SPLINE
SPL {X  -150.342, Y  +330.952, Z    +0.000, E1   +71.154, E3 +35565.120}
SPL {X  -141.358, Y  +310.748, Z    +0.000, E1   +71.233, E3 +35577.826}
SPL {X  -134.330, Y  +298.778, Z    +0.000, E1   +70.323, E3 +35591.673}
SPL {X  -128.957, Y  +290.989, Z    +0.000, E1   +69.528, E3 +35601.038}
SPL {X  -124.846, Y  +285.632, Z    +0.000, E1   +68.906, E3 +35607.502}
SPL {X  -121.783, Y  +281.927, Z    +0.000, E1   +68.403, E3 +35611.934}
SPL {X   -79.219, Y  +246.688, Z    +0.000, E1   +55.887, E3 +35733.440}
ENDSPLINE

SPLINE
SPL {X  -125.038, Y  +285.873, Z    +0.000, E1   +53.023, E3 +35910.481}
SPL {X  -149.949, Y  +329.886, Z    +0.000, E1   +41.515, E3 +35932.046}
SPL {X  -157.246, Y  +356.141, Z    +0.000, E1   +27.282, E3 +35937.103}
SPL {X  -159.525, Y  +373.376, Z    +0.000, E1   +13.812, E3 +35938.760}
SPL {X  -160.000, Y  +387.264, Z    +0.000, E1    +0.544, E3 +35939.218}
SPL {X  -160.000, Y  +390.384, Z    +0.000, E1    -6.008, E3 +35939.255}
SPL {X  -160.000, Y  +395.752, Z    +0.000, E1   -19.038, E3 +35939.449}
SPL {X  -160.000, Y  +404.289, Z    +0.000, E1   -38.292, E3 +35940.117}
SPL {X  -160.000, Y  +418.681, Z    +0.000, E1   -56.949, E3 +35942.307}
SPL {X  -160.000, Y  +471.977, Z    +0.000, E1   -70.792, E3 +35958.826}
SPL {X  -159.977, Y  +677.138, Z    +0.000, E1   -73.665, E3 +36055.317}
SPL {X  -157.805, Y  +700.810, Z    +0.000, E1   -73.511, E3 +36072.147}
SPL {X  -152.242, Y  +723.618, Z    +0.000, E1   -72.940, E3 +36092.060}
SPL {X  -145.929, Y  +740.010, Z    +0.000, E1   -72.229, E3 +36108.532}
SPL {X  -139.114, Y  +753.439, Z    +0.000, E1   -71.436, E3 +36123.170}
SPL {X  -132.333, Y  +764.333, Z    +0.000, E1   -70.535, E3 +36135.794}
SPL {X  -125.486, Y  +773.664, Z    +0.000, E1   -69.598, E3 +36146.768}
SPL {X  -121.321, Y  +778.713, Z    +0.000, E1   -68.872, E3 +36152.778}
SPL {X   -77.337, Y  +814.468, Z    +0.000, E1   -56.377, E3 +36271.410}
ENDSPLINE

SPLINE
SPL {X  -134.727, Y  +760.706, Z    +0.000, E1   -50.460, E3 +36459.641}
SPL {X  -155.580, Y  +711.748, Z    +0.000, E1   -32.084, E3 +36476.556}
SPL {X  -159.445, Y  +687.715, Z    +0.000, E1   -14.660, E3 +36479.403}
SPL {X  -159.995, Y  +675.725, Z    +0.000, E1    -3.424, E3 +36479.914}
SPL {X  -160.000, Y  +671.714, Z    +0.000, E1    +0.835, E3 +36479.954}
SPL {X  -160.000, Y  +663.084, Z    +0.000, E1   +21.134, E3 +36480.278}
SPL {X  -160.000, Y  +650.910, Z    +0.000, E1   +46.005, E3 +36481.432}
SPL {X  -160.000, Y  +634.843, Z    +0.000, E1   +61.273, E3 +36484.109}
SPL {X  -160.000, Y  +578.679, Z    +0.000, E1   +71.665, E3 +36501.943}
SPL {X  -160.000, Y  +387.528, Z    +0.000, E1   +73.487, E3 +36594.755}
SPL {X  -159.218, Y  +369.903, Z    +0.000, E1   +73.425, E3 +36606.622}
SPL {X  -156.808, Y  +353.900, Z    +0.000, E1   +73.180, E3 +36619.226}
SPL {X  -154.539, Y  +344.254, Z    +0.000, E1   +72.827, E3 +36628.763}
ENDSPLINE

SPLINE
SPL {X  -157.258, Y  +356.206, Z    +0.000, E1   +70.434, E3 +36643.336}
ENDSPLINE

SPLINE
SPL {X  -150.342, Y  +330.952, Z    +0.000, E1   +71.154, E3 +36655.008}
SPL {X  -141.358, Y  +310.748, Z    +0.000, E1   +71.233, E3 +36667.714}
SPL {X  -134.330, Y  +298.778, Z    +0.000, E1   +70.323, E3 +36681.561}
SPL {X  -128.957, Y  +290.989, Z    +0.000, E1   +69.528, E3 +36690.926}
SPL {X  -124.846, Y  +285.632, Z    +0.000, E1   +68.906, E3 +36697.390}
SPL {X  -121.783, Y  +281.927, Z    +0.000, E1   +68.403, E3 +36701.822}
SPL {X   -79.219, Y  +246.688, Z    +0.000, E1   +55.887, E3 +36823.328}
ENDSPLINE

SPLINE
SPL {X  -125.038, Y  +285.873, Z    +0.000, E1   +53.023, E3 +37000.369}
SPL {X  -149.949, Y  +329.886, Z    +0.000, E1   +41.515, E3 +37021.934}
SPL {X  -157.246, Y  +356.141, Z    +0.000, E1   +27.282, E3 +37026.991}
SPL {X  -159.525, Y  +373.376, Z    +0.000, E1   +13.812, E3 +37028.648}
SPL {X  -160.000, Y  +387.264, Z    +0.000, E1    +0.544, E3 +37029.106}
SPL {X  -160.000, Y  +390.384, Z    +0.000, E1    -6.008, E3 +37029.143}
SPL {X  -160.000, Y  +395.752, Z    +0.000, E1   -19.038, E3 +37029.337}
SPL {X  -160.000, Y  +404.289, Z    +0.000, E1   -38.292, E3 +37030.005}
SPL {X  -160.000, Y  +418.681, Z    +0.000, E1   -56.949, E3 +37032.195}
SPL {X  -160.000, Y  +471.977, Z    +0.000, E1   -70.792, E3 +37048.714}
SPL {X  -159.977, Y  +677.138, Z    +0.000, E1   -73.665, E3 +37145.205}
SPL {X  -157.805, Y  +700.810, Z    +0.000, E1   -73.511, E3 +37162.035}
SPL {X  -152.242, Y  +723.618, Z    +0.000, E1   -72.940, E3 +37181.948}
SPL {X  -145.929, Y  +740.010, Z    +0.000, E1   -72.229, E3 +37198.420}
SPL {X  -139.114, Y  +753.439, Z    +0.000, E1   -71.436, E3 +37213.058}
SPL {X  -132.333, Y  +764.333, Z    +0.000, E1   -70.535, E3 +37225.682}
SPL {X  -125.486, Y  +773.664, Z    +0.000, E1   -69.598, E3 +37236.656}
SPL {X  -121.321, Y  +778.713, Z    +0.000, E1   -68.872, E3 +37242.666}
SPL {X   -77.337, Y  +814.468, Z    +0.000, E1   -56.377, E3 +37361.298}
ENDSPLINE

SPLINE
SPL {X  -134.727, Y  +760.706, Z    +0.000, E1   -50.460, E3 +37549.529}
SPL {X  -155.580, Y  +711.748, Z    +0.000, E1   -32.084, E3 +37566.444}
SPL {X  -159.445, Y  +687.715, Z    +0.000, E1   -14.660, E3 +37569.291}
SPL {X  -159.995, Y  +675.725, Z    +0.000, E1    -3.424, E3 +37569.802}
SPL {X  -160.000, Y  +671.714, Z    +0.000, E1    +0.835, E3 +37569.842}
SPL {X  -160.000, Y  +663.084, Z    +0.000, E1   +21.134, E3 +37570.166}
SPL {X  -160.000, Y  +650.910, Z    +0.000, E1   +46.005, E3 +37571.320}
SPL {X  -160.000, Y  +634.843, Z    +0.000, E1   +61.273, E3 +37573.997}
SPL {X  -160.000, Y  +578.679, Z    +0.000, E1   +71.665, E3 +37591.831}
SPL {X  -160.000, Y  +387.528, Z    +0.000, E1   +73.487, E3 +37684.643}
SPL {X  -159.218, Y  +369.903, Z    +0.000, E1   +73.425, E3 +37696.510}
SPL {X  -156.808, Y  +353.900, Z    +0.000, E1   +73.180, E3 +37709.114}
SPL {X  -154.539, Y  +344.254, Z    +0.000, E1   +72.827, E3 +37718.651}
ENDSPLINE

SPLINE
SPL {X  -157.258, Y  +356.206, Z    +0.000, E1   +70.434, E3 +37733.224}
ENDSPLINE

SPLINE
SPL {X  -150.342, Y  +330.952, Z    +0.000, E1   +71.154, E3 +37744.896}
SPL {X  -141.358, Y  +310.748, Z    +0.000, E1   +71.233, E3 +37757.602}
SPL {X  -134.330, Y  +298.778, Z    +0.000, E1   +70.323, E3 +37771.449}
SPL {X  -128.957, Y  +290.989, Z    +0.000, E1   +69.528, E3 +37780.814}
SPL {X  -124.846, Y  +285.632, Z    +0.000, E1   +68.906, E3 +37787.278}
SPL {X  -121.783, Y  +281.927, Z    +0.000, E1   +68.403, E3 +37791.710}
SPL {X   -79.219, Y  +246.688, Z    +0.000, E1   +55.887, E3 +37913.216}
ENDSPLINE

SPLINE
SPL {X  -125.038, Y  +285.873, Z    +0.000, E1   +53.023, E3 +38090.257}
SPL {X  -149.949, Y  +329.886, Z    +0.000, E1   +41.515, E3 +38111.822}
SPL {X  -157.246, Y  +356.141, Z    +0.000, E1   +27.282, E3 +38116.879}
SPL {X  -159.525, Y  +373.376, Z    +0.000, E1   +13.812, E3 +38118.536}
SPL {X  -160.000, Y  +387.264, Z    +0.000, E1    +0.544, E3 +38118.994}
SPL {X  -160.000, Y  +390.384, Z    +0.000, E1    -6.008, E3 +38119.031}
SPL {X  -160.000, Y  +395.752, Z    +0.000, E1   -19.038, E3 +38119.225}
SPL {X  -160.000, Y  +404.289, Z    +0.000, E1   -38.292, E3 +38119.893}
SPL {X  -160.000, Y  +418.681, Z    +0.000, E1   -56.949, E3 +38122.083}
SPL {X  -160.000, Y  +471.977, Z    +0.000, E1   -70.792, E3 +38138.602}
SPL {X  -159.977, Y  +677.138, Z    +0.000, E1   -73.665, E3 +38235.093}
SPL {X  -157.805, Y  +700.810, Z    +0.000, E1   -73.511, E3 +38251.923}
SPL {X  -152.242, Y  +723.618, Z    +0.000, E1   -72.940, E3 +38271.836}
SPL {X  -145.929, Y  +740.010, Z    +0.000, E1   -72.229, E3 +38288.308}
SPL {X  -139.114, Y  +753.439, Z    +0.000, E1   -71.436, E3 +38302.946}
SPL {X  -132.333, Y  +764.333, Z    +0.000, E1   -70.535, E3 +38315.570}
SPL {X  -125.486, Y  +773.664, Z    +0.000, E1   -69.598, E3 +38326.544}
SPL {X  -121.321, Y  +778.713, Z    +0.000, E1   -68.872, E3 +38332.554}
SPL {X   -77.337, Y  +814.468, Z    +0.000, E1   -56.377, E3 +38451.186}
ENDSPLINE

SPLINE
SPL {X  -134.727, Y  +760.706, Z    +0.000, E1   -50.460, E3 +38639.417}
SPL {X  -155.580, Y  +711.748, Z    +0.000, E1   -32.084, E3 +38656.332}
SPL {X  -159.445, Y  +687.715, Z    +0.000, E1   -14.660, E3 +38659.179}
SPL {X  -159.995, Y  +675.725, Z    +0.000, E1    -3.424, E3 +38659.690}
SPL {X  -160.000, Y  +671.714, Z    +0.000, E1    +0.835, E3 +38659.730}
SPL {X  -160.000, Y  +663.084, Z    +0.000, E1   +21.134, E3 +38660.054}
SPL {X  -160.000, Y  +650.910, Z    +0.000, E1   +46.005, E3 +38661.208}
SPL {X  -160.000, Y  +634.843, Z    +0.000, E1   +61.273, E3 +38663.885}
SPL {X  -160.000, Y  +578.679, Z    +0.000, E1   +71.665, E3 +38681.719}
SPL {X  -160.000, Y  +387.528, Z    +0.000, E1   +73.487, E3 +38774.531}
SPL {X  -159.218, Y  +369.903, Z    +0.000, E1   +73.425, E3 +38786.398}
SPL {X  -156.808, Y  +353.900, Z    +0.000, E1   +73.180, E3 +38799.002}
SPL {X  -154.539, Y  +344.254, Z    +0.000, E1   +72.827, E3 +38808.539}
ENDSPLINE

SPLINE
SPL {X  -157.258, Y  +356.206, Z    +0.000, E1   +70.434, E3 +38823.112}
ENDSPLINE

SPLINE
SPL {X  -150.342, Y  +330.952, Z    +0.000, E1   +71.154, E3 +38834.784}
SPL {X  -141.358, Y  +310.748, Z    +0.000, E1   +71.233, E3 +38847.490}
SPL {X  -134.330, Y  +298.778, Z    +0.000, E1   +70.323, E3 +38861.337}
SPL {X  -128.957, Y  +290.989, Z    +0.000, E1   +69.528, E3 +38870.702}
SPL {X  -124.846, Y  +285.632, Z    +0.000, E1   +68.906, E3 +38877.166}
SPL {X  -121.783, Y  +281.927, Z    +0.000, E1   +68.403, E3 +38881.598}
SPL {X   -79.219, Y  +246.688, Z    +0.000, E1   +55.887, E3 +39003.104}
ENDSPLINE

SPLINE
SPL {X  -125.038, Y  +285.873, Z    +0.000, E1   +53.023, E3 +39180.145}
SPL {X  -149.949, Y  +329.886, Z    +0.000, E1   +41.515, E3 +39201.710}
SPL {X  -157.246, Y  +356.141, Z    +0.000, E1   +27.282, E3 +39206.767}
SPL {X  -159.525, Y  +373.376, Z    +0.000, E1   +13.812, E3 +39208.424}
SPL {X  -160.000, Y  +387.264, Z    +0.000, E1    +0.544, E3 +39208.882}
SPL {X  -160.000, Y  +390.384, Z    +0.000, E1    -6.008, E3 +39208.919}
SPL {X  -160.000, Y  +395.752, Z    +0.000, E1   -19.038, E3 +39209.113}
SPL {X  -160.000, Y  +404.289, Z    +0.000, E1   -38.292, E3 +39209.781}
SPL {X  -160.000, Y  +418.681, Z    +0.000, E1   -56.949, E3 +39211.971}
SPL {X  -160.000, Y  +471.977, Z    +0.000, E1   -70.792, E3 +39228.490}
SPL {X  -159.977, Y  +677.138, Z    +0.000, E1   -73.665, E3 +39324.981}
SPL {X  -157.805, Y  +700.810, Z    +0.000, E1   -73.511, E3 +39341.812}
SPL {X  -152.242, Y  +723.618, Z    +0.000, E1   -72.940, E3 +39361.724}
SPL {X  -145.929, Y  +740.010, Z    +0.000, E1   -72.229, E3 +39378.196}
SPL {X  -139.114, Y  +753.439, Z    +0.000, E1   -71.436, E3 +39392.834}
SPL {X  -132.333, Y  +764.333, Z    +0.000, E1   -70.535, E3 +39405.458}
SPL {X  -125.486, Y  +773.664, Z    +0.000, E1   -69.598, E3 +39416.432}
SPL {X  -121.321, Y  +778.713, Z    +0.000, E1   -68.872, E3 +39422.442}
SPL {X   -77.337, Y  +814.468, Z    +0.000, E1   -56.377, E3 +39541.074}
ENDSPLINE

SPLINE
SPL {X  -134.727, Y  +760.706, Z    +0.000, E1   -50.460, E3 +39729.306}
SPL {X  -155.580, Y  +711.748, Z    +0.000, E1   -32.084, E3 +39746.220}
SPL {X  -159.445, Y  +687.715, Z    +0.000, E1   -14.660, E3 +39749.067}
SPL {X  -159.995, Y  +675.725, Z    +0.000, E1    -3.424, E3 +39749.578}
SPL {X  -160.000, Y  +671.714, Z    +0.000, E1    +0.835, E3 +39749.618}
SPL {X  -160.000, Y  +663.084, Z    +0.000, E1   +21.134, E3 +39749.943}
SPL {X  -160.000, Y  +650.910, Z    +0.000, E1   +46.005, E3 +39751.096}
SPL {X  -160.000, Y  +634.843, Z    +0.000, E1   +61.273, E3 +39753.773}
SPL {X  -160.000, Y  +578.679, Z    +0.000, E1   +71.665, E3 +39771.607}
SPL {X  -160.000, Y  +387.528, Z    +0.000, E1   +73.487, E3 +39864.419}
SPL {X  -159.218, Y  +369.903, Z    +0.000, E1   +73.425, E3 +39876.286}
SPL {X  -156.808, Y  +353.900, Z    +0.000, E1   +73.180, E3 +39888.890}
SPL {X  -154.539, Y  +344.254, Z    +0.000, E1   +72.827, E3 +39898.428}
ENDSPLINE

SPLINE
SPL {X  -157.258, Y  +356.206, Z    +0.000, E1   +70.434, E3 +39913.000}
ENDSPLINE

SPLINE
SPL {X  -150.342, Y  +330.952, Z    +0.000, E1   +71.154, E3 +39924.672}
SPL {X  -141.358, Y  +310.748, Z    +0.000, E1   +71.233, E3 +39937.378}
SPL {X  -134.330, Y  +298.778, Z    +0.000, E1   +70.323, E3 +39951.225}
SPL {X  -128.957, Y  +290.989, Z    +0.000, E1   +69.528, E3 +39960.591}
SPL {X  -124.846, Y  +285.632, Z    +0.000, E1   +68.906, E3 +39967.054}
SPL {X  -121.783, Y  +281.927, Z    +0.000, E1   +68.403, E3 +39971.486}
SPL {X   -79.219, Y  +246.688, Z    +0.000, E1   +55.887, E3 +40092.992}
ENDSPLINE

SPLINE
SPL {X  -125.038, Y  +285.873, Z    +0.000, E1   +53.023, E3 +40270.033}
SPL {X  -149.949, Y  +329.886, Z    +0.000, E1   +41.515, E3 +40291.599}
SPL {X  -157.246, Y  +356.141, Z    +0.000, E1   +27.282, E3 +40296.655}
SPL {X  -159.525, Y  +373.376, Z    +0.000, E1   +13.812, E3 +40298.312}
SPL {X  -160.000, Y  +387.264, Z    +0.000, E1    +0.544, E3 +40298.770}
SPL {X  -160.000, Y  +390.384, Z    +0.000, E1    -6.008, E3 +40298.807}
SPL {X  -160.000, Y  +395.752, Z    +0.000, E1   -19.038, E3 +40299.001}
SPL {X  -160.000, Y  +404.289, Z    +0.000, E1   -38.292, E3 +40299.669}
SPL {X  -160.000, Y  +418.681, Z    +0.000, E1   -56.949, E3 +40301.859}
SPL {X  -160.000, Y  +471.977, Z    +0.000, E1   -70.792, E3 +40318.378}
SPL {X  -159.977, Y  +677.138, Z    +0.000, E1   -73.665, E3 +40414.869}
SPL {X  -157.805, Y  +700.810, Z    +0.000, E1   -73.511, E3 +40431.700}
SPL {X  -152.242, Y  +723.618, Z    +0.000, E1   -72.940, E3 +40451.612}
SPL {X  -145.929, Y  +740.010, Z    +0.000, E1   -72.229, E3 +40468.084}
SPL {X  -139.114, Y  +753.439, Z    +0.000, E1   -71.436, E3 +40482.722}
SPL {X  -132.333, Y  +764.333, Z    +0.000, E1   -70.535, E3 +40495.346}
SPL {X  -125.486, Y  +773.664, Z    +0.000, E1   -69.598, E3 +40506.320}
SPL {X  -121.321, Y  +778.713, Z    +0.000, E1   -68.872, E3 +40512.330}
SPL {X   -77.337, Y  +814.468, Z    +0.000, E1   -56.377, E3 +40630.962}
ENDSPLINE

SPLINE
SPL {X  -134.727, Y  +760.706, Z    +0.000, E1   -50.460, E3 +40819.194}
SPL {X  -155.580, Y  +711.748, Z    +0.000, E1   -32.084, E3 +40836.108}
SPL {X  -159.445, Y  +687.715, Z    +0.000, E1   -14.660, E3 +40838.955}
SPL {X  -159.995, Y  +675.725, Z    +0.000, E1    -3.424, E3 +40839.466}
SPL {X  -160.000, Y  +671.714, Z    +0.000, E1    +0.835, E3 +40839.506}
SPL {X  -160.000, Y  +663.084, Z    +0.000, E1   +21.134, E3 +40839.831}
SPL {X  -160.000, Y  +650.910, Z    +0.000, E1   +46.005, E3 +40840.984}
SPL {X  -160.000, Y  +634.843, Z    +0.000, E1   +61.273, E3 +40843.661}
SPL {X  -160.000, Y  +578.679, Z    +0.000, E1   +71.665, E3 +40861.495}
SPL {X  -160.000, Y  +387.528, Z    +0.000, E1   +73.487, E3 +40954.307}
SPL {X  -159.218, Y  +369.903, Z    +0.000, E1   +73.425, E3 +40966.175}
SPL {X  -156.808, Y  +353.900, Z    +0.000, E1   +73.180, E3 +40978.778}
SPL {X  -154.539, Y  +344.254, Z    +0.000, E1   +72.827, E3 +40988.316}
ENDSPLINE

SPLINE
SPL {X  -157.258, Y  +356.206, Z    +0.000, E1   +70.434, E3 +41002.888}
ENDSPLINE

SPLINE
SPL {X  -150.342, Y  +330.952, Z    +0.000, E1   +71.154, E3 +41014.560}
SPL {X  -141.358, Y  +310.748, Z    +0.000, E1   +71.233, E3 +41027.266}
SPL {X  -134.330, Y  +298.778, Z    +0.000, E1   +70.323, E3 +41041.113}
SPL {X  -128.957, Y  +290.989, Z    +0.000, E1   +69.528, E3 +41050.479}
SPL {X  -124.846, Y  +285.632, Z    +0.000, E1   +68.906, E3 +41056.942}
SPL {X  -121.783, Y  +281.927, Z    +0.000, E1   +68.403, E3 +41061.374}
SPL {X   -79.219, Y  +246.688, Z    +0.000, E1   +55.887, E3 +41182.880}
ENDSPLINE

SPLINE
SPL {X  -125.038, Y  +285.873, Z    +0.000, E1   +53.023, E3 +41359.921}
SPL {X  -149.949, Y  +329.886, Z    +0.000, E1   +41.515, E3 +41381.487}
SPL {X  -157.246, Y  +356.141, Z    +0.000, E1   +27.282, E3 +41386.543}
SPL {X  -159.525, Y  +373.376, Z    +0.000, E1   +13.812, E3 +41388.200}
SPL {X  -160.000, Y  +387.264, Z    +0.000, E1    +0.544, E3 +41388.658}
SPL {X  -160.000, Y  +390.384, Z    +0.000, E1    -6.008, E3 +41388.695}
SPL {X  -160.000, Y  +395.752, Z    +0.000, E1   -19.038, E3 +41388.889}
SPL {X  -160.000, Y  +404.289, Z    +0.000, E1   -38.292, E3 +41389.557}
SPL {X  -160.000, Y  +418.681, Z    +0.000, E1   -56.949, E3 +41391.747}
SPL {X  -160.000, Y  +471.977, Z    +0.000, E1   -70.792, E3 +41408.266}
SPL {X  -159.977, Y  +677.138, Z    +0.000, E1   -73.665, E3 +41504.757}
SPL {X  -157.805, Y  +700.810, Z    +0.000, E1   -73.511, E3 +41521.588}
SPL {X  -152.242, Y  +723.618, Z    +0.000, E1   -72.940, E3 +41541.500}
SPL {X  -145.929, Y  +740.010, Z    +0.000, E1   -72.229, E3 +41557.972}
SPL {X  -139.114, Y  +753.439, Z    +0.000, E1   -71.436, E3 +41572.611}
SPL {X  -132.333, Y  +764.333, Z    +0.000, E1   -70.535, E3 +41585.234}
SPL {X  -125.486, Y  +773.664, Z    +0.000, E1   -69.598, E3 +41596.209}
SPL {X  -121.321, Y  +778.713, Z    +0.000, E1   -68.872, E3 +41602.219}
SPL {X   -77.337, Y  +814.468, Z    +0.000, E1   -56.377, E3 +41720.850}
ENDSPLINE

SPLINE
SPL {X  -134.727, Y  +760.706, Z    +0.000, E1   -50.460, E3 +41909.082}
SPL {X  -155.580, Y  +711.748, Z    +0.000, E1   -32.084, E3 +41925.996}
SPL {X  -159.445, Y  +687.715, Z    +0.000, E1   -14.660, E3 +41928.843}
SPL {X  -159.995, Y  +675.725, Z    +0.000, E1    -3.424, E3 +41929.354}
SPL {X  -160.000, Y  +671.714, Z    +0.000, E1    +0.835, E3 +41929.394}
SPL {X  -160.000, Y  +663.084, Z    +0.000, E1   +21.134, E3 +41929.719}
SPL {X  -160.000, Y  +650.910, Z    +0.000, E1   +46.005, E3 +41930.872}
SPL {X  -160.000, Y  +634.843, Z    +0.000, E1   +61.273, E3 +41933.549}
SPL {X  -160.000, Y  +578.679, Z    +0.000, E1   +71.665, E3 +41951.383}
SPL {X  -160.000, Y  +387.528, Z    +0.000, E1   +73.487, E3 +42044.195}
SPL {X  -159.218, Y  +369.903, Z    +0.000, E1   +73.425, E3 +42056.063}
SPL {X  -156.808, Y  +353.900, Z    +0.000, E1   +73.180, E3 +42068.666}
SPL {X  -154.539, Y  +344.254, Z    +0.000, E1   +72.827, E3 +42078.204}
ENDSPLINE

SPLINE
SPL {X  -157.258, Y  +356.206, Z    +0.000, E1   +70.434, E3 +42092.776}
ENDSPLINE

SPLINE
SPL {X  -150.342, Y  +330.952, Z    +0.000, E1   +71.154, E3 +42104.448}
SPL {X  -141.358, Y  +310.748, Z    +0.000, E1   +71.233, E3 +42117.154}
SPL {X  -134.330, Y  +298.778, Z    +0.000, E1   +70.323, E3 +42131.001}
SPL {X  -128.957, Y  +290.989, Z    +0.000, E1   +69.528, E3 +42140.367}
SPL {X  -124.846, Y  +285.632, Z    +0.000, E1   +68.906, E3 +42146.830}
SPL {X  -121.783, Y  +281.927, Z    +0.000, E1   +68.403, E3 +42151.262}
SPL {X   -79.219, Y  +246.688, Z    +0.000, E1   +55.887, E3 +42272.768}
ENDSPLINE

SPLINE
SPL {X  -125.038, Y  +285.873, Z    +0.000, E1   +53.023, E3 +42449.810}
SPL {X  -149.949, Y  +329.886, Z    +0.000, E1   +41.515, E3 +42471.375}
SPL {X  -157.246, Y  +356.141, Z    +0.000, E1   +27.282, E3 +42476.431}
SPL {X  -159.525, Y  +373.376, Z    +0.000, E1   +13.812, E3 +42478.088}
SPL {X  -160.000, Y  +387.264, Z    +0.000, E1    +0.544, E3 +42478.546}
SPL {X  -160.000, Y  +390.384, Z    +0.000, E1    -6.008, E3 +42478.583}
SPL {X  -160.000, Y  +395.752, Z    +0.000, E1   -19.038, E3 +42478.777}
SPL {X  -160.000, Y  +404.289, Z    +0.000, E1   -38.292, E3 +42479.445}
SPL {X  -160.000, Y  +418.681, Z    +0.000, E1   -56.949, E3 +42481.635}
SPL {X  -160.000, Y  +471.977, Z    +0.000, E1   -70.792, E3 +42498.154}
SPL {X  -159.977, Y  +677.138, Z    +0.000, E1   -73.665, E3 +42594.645}
SPL {X  -157.805, Y  +700.810, Z    +0.000, E1   -73.511, E3 +42611.476}
SPL {X  -152.242, Y  +723.618, Z    +0.000, E1   -72.940, E3 +42631.389}
SPL {X  -145.929, Y  +740.010, Z    +0.000, E1   -72.229, E3 +42647.860}
SPL {X  -139.114, Y  +753.439, Z    +0.000, E1   -71.436, E3 +42662.499}
SPL {X  -132.333, Y  +764.333, Z    +0.000, E1   -70.535, E3 +42675.122}
SPL {X  -125.486, Y  +773.664, Z    +0.000, E1   -69.598, E3 +42686.097}
SPL {X  -121.321, Y  +778.713, Z    +0.000, E1   -68.872, E3 +42692.107}
SPL {X   -77.337, Y  +814.468, Z    +0.000, E1   -56.377, E3 +42810.738}
ENDSPLINE

SPLINE
SPL {X  -134.727, Y  +760.706, Z    +0.000, E1   -50.460, E3 +42998.970}
SPL {X  -155.580, Y  +711.748, Z    +0.000, E1   -32.084, E3 +43015.884}
SPL {X  -159.445, Y  +687.715, Z    +0.000, E1   -14.660, E3 +43018.731}
SPL {X  -159.995, Y  +675.725, Z    +0.000, E1    -3.424, E3 +43019.242}
SPL {X  -160.000, Y  +671.714, Z    +0.000, E1    +0.835, E3 +43019.282}
SPL {X  -160.000, Y  +663.084, Z    +0.000, E1   +21.134, E3 +43019.607}
SPL {X  -160.000, Y  +650.910, Z    +0.000, E1   +46.005, E3 +43020.760}
SPL {X  -160.000, Y  +634.843, Z    +0.000, E1   +61.273, E3 +43023.437}
SPL {X  -160.000, Y  +578.679, Z    +0.000, E1   +71.665, E3 +43041.271}
SPL {X  -160.000, Y  +387.528, Z    +0.000, E1   +73.487, E3 +43134.083}
SPL {X  -159.218, Y  +369.903, Z    +0.000, E1   +73.425, E3 +43145.951}
SPL {X  -156.808, Y  +353.900, Z    +0.000, E1   +73.180, E3 +43158.554}
SPL {X  -154.539, Y  +344.254, Z    +0.000, E1   +72.827, E3 +43168.092}
ENDSPLINE

SPLINE
SPL {X  -157.258, Y  +356.206, Z    +0.000, E1   +70.434, E3 +43182.664}
ENDSPLINE

SPLINE
SPL {X  -150.342, Y  +330.952, Z    +0.000, E1   +71.154, E3 +43194.336}
SPL {X  -141.358, Y  +310.748, Z    +0.000, E1   +71.233, E3 +43207.042}
SPL {X  -134.330, Y  +298.778, Z    +0.000, E1   +70.323, E3 +43220.889}
SPL {X  -128.957, Y  +290.989, Z    +0.000, E1   +69.528, E3 +43230.255}
SPL {X  -124.846, Y  +285.632, Z    +0.000, E1   +68.906, E3 +43236.718}
SPL {X  -121.783, Y  +281.927, Z    +0.000, E1   +68.403, E3 +43241.150}
SPL {X   -79.219, Y  +246.688, Z    +0.000, E1   +55.887, E3 +43362.656}
ENDSPLINE

SPLINE
SPL {X  -125.038, Y  +285.873, Z    +0.000, E1   +53.023, E3 +43539.698}
SPL {X  -149.949, Y  +329.886, Z    +0.000, E1   +41.515, E3 +43561.263}
SPL {X  -157.246, Y  +356.141, Z    +0.000, E1   +27.282, E3 +43566.319}
SPL {X  -159.525, Y  +373.376, Z    +0.000, E1   +13.812, E3 +43567.976}
SPL {X  -160.000, Y  +387.264, Z    +0.000, E1    +0.544, E3 +43568.434}
SPL {X  -160.000, Y  +390.384, Z    +0.000, E1    -6.008, E3 +43568.471}
SPL {X  -160.000, Y  +395.752, Z    +0.000, E1   -19.038, E3 +43568.665}
SPL {X  -160.000, Y  +404.289, Z    +0.000, E1   -38.292, E3 +43569.333}
SPL {X  -160.000, Y  +418.681, Z    +0.000, E1   -56.949, E3 +43571.523}
SPL {X  -160.000, Y  +471.977, Z    +0.000, E1   -70.792, E3 +43588.042}
SPL {X  -159.977, Y  +677.138, Z    +0.000, E1   -73.665, E3 +43684.533}
SPL {X  -157.805, Y  +700.810, Z    +0.000, E1   -73.511, E3 +43701.364}
SPL {X  -152.242, Y  +723.618, Z    +0.000, E1   -72.940, E3 +43721.277}
SPL {X  -145.929, Y  +740.010, Z    +0.000, E1   -72.229, E3 +43737.748}
SPL {X  -139.114, Y  +753.439, Z    +0.000, E1   -71.436, E3 +43752.387}
SPL {X  -132.333, Y  +764.333, Z    +0.000, E1   -70.535, E3 +43765.010}
SPL {X  -125.486, Y  +773.664, Z    +0.000, E1   -69.598, E3 +43775.985}
SPL {X  -121.321, Y  +778.713, Z    +0.000, E1   -68.872, E3 +43781.995}
SPL {X   -77.337, Y  +814.468, Z    +0.000, E1   -56.377, E3 +43900.626}
ENDSPLINE

SPLINE
SPL {X  -134.727, Y  +760.706, Z    +0.000, E1   -50.460, E3 +44088.858}
SPL {X  -155.580, Y  +711.748, Z    +0.000, E1   -32.084, E3 +44105.772}
SPL {X  -159.445, Y  +687.715, Z    +0.000, E1   -14.660, E3 +44108.619}
SPL {X  -159.995, Y  +675.725, Z    +0.000, E1    -3.424, E3 +44109.130}
SPL {X  -160.000, Y  +671.714, Z    +0.000, E1    +0.835, E3 +44109.170}
SPL {X  -160.000, Y  +663.084, Z    +0.000, E1   +21.134, E3 +44109.495}
SPL {X  -160.000, Y  +650.910, Z    +0.000, E1   +46.005, E3 +44110.648}
SPL {X  -160.000, Y  +634.843, Z    +0.000, E1   +61.273, E3 +44113.325}
SPL {X  -160.000, Y  +578.679, Z    +0.000, E1   +71.665, E3 +44131.159}
SPL {X  -160.000, Y  +387.528, Z    +0.000, E1   +73.487, E3 +44223.971}
SPL {X  -159.218, Y  +369.903, Z    +0.000, E1   +73.425, E3 +44235.839}
SPL {X  -156.808, Y  +353.900, Z    +0.000, E1   +73.180, E3 +44248.442}
SPL {X  -154.539, Y  +344.254, Z    +0.000, E1   +72.827, E3 +44257.980}
ENDSPLINE

SPLINE
SPL {X  -157.258, Y  +356.206, Z    +0.000, E1   +70.434, E3 +44272.552}
ENDSPLINE

SPLINE
SPL {X  -150.342, Y  +330.952, Z    +0.000, E1   +71.154, E3 +44284.224}
SPL {X  -141.358, Y  +310.748, Z    +0.000, E1   +71.233, E3 +44296.930}
SPL {X  -134.330, Y  +298.778, Z    +0.000, E1   +70.323, E3 +44310.777}
SPL {X  -128.957, Y  +290.989, Z    +0.000, E1   +69.528, E3 +44320.143}
SPL {X  -124.846, Y  +285.632, Z    +0.000, E1   +68.906, E3 +44326.606}
SPL {X  -121.783, Y  +281.927, Z    +0.000, E1   +68.403, E3 +44331.038}
SPL {X   -79.219, Y  +246.688, Z    +0.000, E1   +55.887, E3 +44452.544}
ENDSPLINE

SPLINE
SPL {X  -125.038, Y  +285.873, Z    +0.000, E1   +53.023, E3 +44629.586}
SPL {X  -149.949, Y  +329.886, Z    +0.000, E1   +41.515, E3 +44651.151}
SPL {X  -157.246, Y  +356.141, Z    +0.000, E1   +27.282, E3 +44656.207}
SPL {X  -159.525, Y  +373.376, Z    +0.000, E1   +13.812, E3 +44657.864}
SPL {X  -160.000, Y  +387.264, Z    +0.000, E1    +0.544, E3 +44658.322}
SPL {X  -160.000, Y  +390.384, Z    +0.000, E1    -6.008, E3 +44658.359}
SPL {X  -160.000, Y  +395.752, Z    +0.000, E1   -19.038, E3 +44658.553}
SPL {X  -160.000, Y  +404.289, Z    +0.000, E1   -38.292, E3 +44659.221}
SPL {X  -160.000, Y  +418.681, Z    +0.000, E1   -56.949, E3 +44661.411}
SPL {X  -160.000, Y  +471.977, Z    +0.000, E1   -70.792, E3 +44677.930}
SPL {X  -159.977, Y  +677.138, Z    +0.000, E1   -73.665, E3 +44774.422}
SPL {X  -157.805, Y  +700.810, Z    +0.000, E1   -73.511, E3 +44791.252}
SPL {X  -152.242, Y  +723.618, Z    +0.000, E1   -72.940, E3 +44811.165}
SPL {X  -145.929, Y  +740.010, Z    +0.000, E1   -72.229, E3 +44827.636}
SPL {X  -139.114, Y  +753.439, Z    +0.000, E1   -71.436, E3 +44842.275}
SPL {X  -132.333, Y  +764.333, Z    +0.000, E1   -70.535, E3 +44854.898}
SPL {X  -125.486, Y  +773.664, Z    +0.000, E1   -69.598, E3 +44865.873}
SPL {X  -121.321, Y  +778.713, Z    +0.000, E1   -68.872, E3 +44871.883}
SPL {X   -77.337, Y  +814.468, Z    +0.000, E1   -56.377, E3 +44990.514}
ENDSPLINE

SPLINE
SPL {X  -134.727, Y  +760.706, Z    +0.000, E1   -50.460, E3 +45178.746}
SPL {X  -155.580, Y  +711.748, Z    +0.000, E1   -32.084, E3 +45195.660}
SPL {X  -159.445, Y  +687.715, Z    +0.000, E1   -14.660, E3 +45198.507}
SPL {X  -159.995, Y  +675.725, Z    +0.000, E1    -3.424, E3 +45199.018}
SPL {X  -160.000, Y  +671.714, Z    +0.000, E1    +0.835, E3 +45199.058}
SPL {X  -160.000, Y  +663.084, Z    +0.000, E1   +21.134, E3 +45199.383}
SPL {X  -160.000, Y  +650.910, Z    +0.000, E1   +46.005, E3 +45200.536}
SPL {X  -160.000, Y  +634.843, Z    +0.000, E1   +61.273, E3 +45203.213}
SPL {X  -160.000, Y  +578.679, Z    +0.000, E1   +71.665, E3 +45221.047}
SPL {X  -160.000, Y  +387.528, Z    +0.000, E1   +73.487, E3 +45313.859}
SPL {X  -159.218, Y  +369.903, Z    +0.000, E1   +73.425, E3 +45325.727}
SPL {X  -156.808, Y  +353.900, Z    +0.000, E1   +73.180, E3 +45338.330}
SPL {X  -154.539, Y  +344.254, Z    +0.000, E1   +72.827, E3 +45347.868}
ENDSPLINE

SPLINE
SPL {X  -157.258, Y  +356.206, Z    +0.000, E1   +70.434, E3 +45362.440}
ENDSPLINE

SPLINE
SPL {X  -150.342, Y  +330.952, Z    +0.000, E1   +71.154, E3 +45374.113}
SPL {X  -141.358, Y  +310.748, Z    +0.000, E1   +71.233, E3 +45386.818}
SPL {X  -134.330, Y  +298.778, Z    +0.000, E1   +70.323, E3 +45400.666}
SPL {X  -128.957, Y  +290.989, Z    +0.000, E1   +69.528, E3 +45410.031}
SPL {X  -124.846, Y  +285.632, Z    +0.000, E1   +68.906, E3 +45416.494}
SPL {X  -121.783, Y  +281.927, Z    +0.000, E1   +68.403, E3 +45420.926}
SPL {X   -79.219, Y  +246.688, Z    +0.000, E1   +55.887, E3 +45542.433}
ENDSPLINE

SPLINE
SPL {X  -125.038, Y  +285.873, Z    +0.000, E1   +53.023, E3 +45719.474}
SPL {X  -149.949, Y  +329.886, Z    +0.000, E1   +41.515, E3 +45741.039}
SPL {X  -157.246, Y  +356.141, Z    +0.000, E1   +27.282, E3 +45746.095}
SPL {X  -159.525, Y  +373.376, Z    +0.000, E1   +13.812, E3 +45747.752}
SPL {X  -160.000, Y  +387.264, Z    +0.000, E1    +0.544, E3 +45748.210}
SPL {X  -160.000, Y  +390.384, Z    +0.000, E1    -6.008, E3 +45748.247}
SPL {X  -160.000, Y  +395.752, Z    +0.000, E1   -19.038, E3 +45748.441}
SPL {X  -160.000, Y  +404.289, Z    +0.000, E1   -38.292, E3 +45749.109}
SPL {X  -160.000, Y  +418.681, Z    +0.000, E1   -56.949, E3 +45751.299}
SPL {X  -160.000, Y  +458.961, Z    +0.000, E1   -69.778, E3 +45762.896}
SPL {X  -160.000, Y  +485.343, Z    +0.000, E1   -71.539, E3 +45772.881}
SPL {X  -159.977, Y  +677.138, Z    +0.000, E1   -73.665, E3 +45864.310}
SPL {X  -157.805, Y  +700.810, Z    +0.000, E1   -73.511, E3 +45881.140}
SPL {X  -152.242, Y  +723.618, Z    +0.000, E1   -72.940, E3 +45901.053}
SPL {X  -145.929, Y  +740.010, Z    +0.000, E1   -72.229, E3 +45917.524}
SPL {X  -139.114, Y  +753.439, Z    +0.000, E1   -71.436, E3 +45932.163}
SPL {X  -132.333, Y  +764.333, Z    +0.000, E1   -70.535, E3 +45944.787}
SPL {X  -125.486, Y  +773.664, Z    +0.000, E1   -69.598, E3 +45955.761}
SPL {X  -121.321, Y  +778.713, Z    +0.000, E1   -68.872, E3 +45961.771}
SPL {X   -77.337, Y  +814.468, Z    +0.000, E1   -56.377, E3 +46080.402}
ENDSPLINE

SPLINE
SPL {X  -134.727, Y  +760.706, Z    +0.000, E1   -50.460, E3 +46268.634}
SPL {X  -155.580, Y  +711.748, Z    +0.000, E1   -32.084, E3 +46285.548}
SPL {X  -159.445, Y  +687.715, Z    +0.000, E1   -14.660, E3 +46288.395}
SPL {X  -159.995, Y  +675.725, Z    +0.000, E1    -3.424, E3 +46288.906}
SPL {X  -160.000, Y  +671.714, Z    +0.000, E1    +0.835, E3 +46288.946}
SPL {X  -160.000, Y  +663.084, Z    +0.000, E1   +21.134, E3 +46289.271}
SPL {X  -160.000, Y  +650.910, Z    +0.000, E1   +46.005, E3 +46290.425}
SPL {X  -160.000, Y  +634.843, Z    +0.000, E1   +61.273, E3 +46293.101}
SPL {X  -160.000, Y  +578.679, Z    +0.000, E1   +71.665, E3 +46310.935}
SPL {X  -160.000, Y  +387.528, Z    +0.000, E1   +73.487, E3 +46403.748}
SPL {X  -159.218, Y  +369.903, Z    +0.000, E1   +73.425, E3 +46415.615}
SPL {X  -156.808, Y  +353.900, Z    +0.000, E1   +73.180, E3 +46428.218}
SPL {X  -154.539, Y  +344.254, Z    +0.000, E1   +72.827, E3 +46437.756}
ENDSPLINE

SPLINE
SPL {X  -157.258, Y  +356.206, Z    +0.000, E1   +70.434, E3 +46452.328}
ENDSPLINE

SPLINE
SPL {X  -150.342, Y  +330.952, Z    +0.000, E1   +71.154, E3 +46464.001}
SPL {X  -141.358, Y  +310.748, Z    +0.000, E1   +71.233, E3 +46476.706}
SPL {X  -134.330, Y  +298.778, Z    +0.000, E1   +70.323, E3 +46490.554}
SPL {X  -128.957, Y  +290.989, Z    +0.000, E1   +69.528, E3 +46499.919}
SPL {X  -124.846, Y  +285.632, Z    +0.000, E1   +68.906, E3 +46506.382}
SPL {X  -121.783, Y  +281.927, Z    +0.000, E1   +68.403, E3 +46510.814}
SPL {X   -79.219, Y  +246.688, Z    +0.000, E1   +55.887, E3 +46632.321}
ENDSPLINE

SPLINE
SPL {X  -125.038, Y  +285.873, Z    +0.000, E1   +53.023, E3 +46809.362}
SPL {X  -149.949, Y  +329.886, Z    +0.000, E1   +41.515, E3 +46830.927}
SPL {X  -157.246, Y  +356.141, Z    +0.000, E1   +27.282, E3 +46835.983}
SPL {X  -159.525, Y  +373.376, Z    +0.000, E1   +13.812, E3 +46837.641}
SPL {X  -160.000, Y  +387.264, Z    +0.000, E1    +0.544, E3 +46838.098}
SPL {X  -160.000, Y  +390.384, Z    +0.000, E1    -6.008, E3 +46838.135}
SPL {X  -160.000, Y  +395.752, Z    +0.000, E1   -19.038, E3 +46838.329}
SPL {X  -160.000, Y  +404.289, Z    +0.000, E1   -38.292, E3 +46838.997}
SPL {X  -160.000, Y  +418.681, Z    +0.000, E1   -56.949, E3 +46841.187}
SPL {X  -160.000, Y  +471.977, Z    +0.000, E1   -70.792, E3 +46857.707}
SPL {X  -159.977, Y  +677.138, Z    +0.000, E1   -73.665, E3 +46954.198}
SPL {X  -157.805, Y  +700.810, Z    +0.000, E1   -73.511, E3 +46971.028}
SPL {X  -152.242, Y  +723.618, Z    +0.000, E1   -72.940, E3 +46990.941}
SPL {X  -145.929, Y  +740.010, Z    +0.000, E1   -72.229, E3 +47007.412}
SPL {X  -139.114, Y  +753.439, Z    +0.000, E1   -71.436, E3 +47022.051}
SPL {X  -132.333, Y  +764.333, Z    +0.000, E1   -70.535, E3 +47034.675}
SPL {X  -125.486, Y  +773.664, Z    +0.000, E1   -69.598, E3 +47045.649}
SPL {X  -121.321, Y  +778.713, Z    +0.000, E1   -68.872, E3 +47051.659}
SPL {X   -77.337, Y  +814.468, Z    +0.000, E1   -56.377, E3 +47170.290}
ENDSPLINE

SPLINE
SPL {X  -134.727, Y  +760.706, Z    +0.000, E1   -50.460, E3 +47358.522}
SPL {X  -155.580, Y  +711.748, Z    +0.000, E1   -32.084, E3 +47375.436}
SPL {X  -159.445, Y  +687.715, Z    +0.000, E1   -14.660, E3 +47378.283}
SPL {X  -159.995, Y  +675.725, Z    +0.000, E1    -3.424, E3 +47378.794}
SPL {X  -160.000, Y  +671.714, Z    +0.000, E1    +0.835, E3 +47378.834}
SPL {X  -160.000, Y  +663.084, Z    +0.000, E1   +21.134, E3 +47379.159}
SPL {X  -160.000, Y  +650.910, Z    +0.000, E1   +46.005, E3 +47380.313}
SPL {X  -160.000, Y  +634.843, Z    +0.000, E1   +61.273, E3 +47382.989}
SPL {X  -160.000, Y  +578.679, Z    +0.000, E1   +71.665, E3 +47400.823}
SPL {X  -160.000, Y  +387.528, Z    +0.000, E1   +73.487, E3 +47493.636}
SPL {X  -159.218, Y  +369.903, Z    +0.000, E1   +73.425, E3 +47505.503}
SPL {X  -156.808, Y  +353.900, Z    +0.000, E1   +73.180, E3 +47518.107}
SPL {X  -154.539, Y  +344.254, Z    +0.000, E1   +72.827, E3 +47527.644}
ENDSPLINE

SPLINE
SPL {X  -157.258, Y  +356.206, Z    +0.000, E1   +70.434, E3 +47542.216}
ENDSPLINE

SPLINE
SPL {X  -150.342, Y  +330.952, Z    +0.000, E1   +71.154, E3 +47553.889}
SPL {X  -141.358, Y  +310.748, Z    +0.000, E1   +71.233, E3 +47566.594}
SPL {X  -134.330, Y  +298.778, Z    +0.000, E1   +70.323, E3 +47580.442}
SPL {X  -128.957, Y  +290.989, Z    +0.000, E1   +69.528, E3 +47589.807}
SPL {X  -124.846, Y  +285.632, Z    +0.000, E1   +68.906, E3 +47596.270}
SPL {X  -121.783, Y  +281.927, Z    +0.000, E1   +68.403, E3 +47600.702}
SPL {X   -79.219, Y  +246.688, Z    +0.000, E1   +55.887, E3 +47722.209}
ENDSPLINE

SPLINE
SPL {X  -125.038, Y  +285.873, Z    +0.000, E1   +53.023, E3 +47899.250}
SPL {X  -149.949, Y  +329.886, Z    +0.000, E1   +41.515, E3 +47920.815}
SPL {X  -157.246, Y  +356.141, Z    +0.000, E1   +27.282, E3 +47925.871}
SPL {X  -159.525, Y  +373.376, Z    +0.000, E1   +13.812, E3 +47927.529}
SPL {X  -160.000, Y  +387.264, Z    +0.000, E1    +0.544, E3 +47927.986}
SPL {X  -160.000, Y  +390.384, Z    +0.000, E1    -6.008, E3 +47928.023}
SPL {X  -160.000, Y  +395.752, Z    +0.000, E1   -19.038, E3 +47928.217}
SPL {X  -160.000, Y  +404.289, Z    +0.000, E1   -38.292, E3 +47928.886}
SPL {X  -160.000, Y  +418.681, Z    +0.000, E1   -56.949, E3 +47931.075}
SPL {X  -160.000, Y  +471.977, Z    +0.000, E1   -70.792, E3 +47947.595}
SPL {X  -159.977, Y  +677.138, Z    +0.000, E1   -73.665, E3 +48044.086}
SPL {X  -157.805, Y  +700.810, Z    +0.000, E1   -73.511, E3 +48060.916}
SPL {X  -152.242, Y  +723.618, Z    +0.000, E1   -72.940, E3 +48080.829}
SPL {X  -145.929, Y  +740.010, Z    +0.000, E1   -72.229, E3 +48097.300}
SPL {X  -139.114, Y  +753.439, Z    +0.000, E1   -71.436, E3 +48111.939}
SPL {X  -132.333, Y  +764.333, Z    +0.000, E1   -70.535, E3 +48124.563}
SPL {X  -125.486, Y  +773.664, Z    +0.000, E1   -69.598, E3 +48135.537}
SPL {X  -121.321, Y  +778.713, Z    +0.000, E1   -68.872, E3 +48141.547}
SPL {X   -77.337, Y  +814.468, Z    +0.000, E1   -56.377, E3 +48260.178}
ENDSPLINE

SPLINE
SPL {X  -134.727, Y  +760.706, Z    +0.000, E1   -50.460, E3 +48448.410}
SPL {X  -155.580, Y  +711.748, Z    +0.000, E1   -32.084, E3 +48465.325}
SPL {X  -159.445, Y  +687.715, Z    +0.000, E1   -14.660, E3 +48468.171}
SPL {X  -159.995, Y  +675.725, Z    +0.000, E1    -3.424, E3 +48468.682}
SPL {X  -160.000, Y  +671.714, Z    +0.000, E1    +0.835, E3 +48468.723}
SPL {X  -160.000, Y  +663.084, Z    +0.000, E1   +21.134, E3 +48469.047}
SPL {X  -160.000, Y  +650.910, Z    +0.000, E1   +46.005, E3 +48470.201}
SPL {X  -160.000, Y  +634.843, Z    +0.000, E1   +61.273, E3 +48472.877}
SPL {X  -160.000, Y  +578.679, Z    +0.000, E1   +71.665, E3 +48490.711}
SPL {X  -160.000, Y  +387.528, Z    +0.000, E1   +73.487, E3 +48583.524}
SPL {X  -159.218, Y  +369.903, Z    +0.000, E1   +73.425, E3 +48595.391}
SPL {X  -156.808, Y  +353.900, Z    +0.000, E1   +73.180, E3 +48607.995}
SPL {X  -154.539, Y  +344.254, Z    +0.000, E1   +72.827, E3 +48617.532}
ENDSPLINE

SPLINE
SPL {X  -157.258, Y  +356.206, Z    +0.000, E1   +70.434, E3 +48632.104}
ENDSPLINE

SPLINE
SPL {X  -150.342, Y  +330.952, Z    +0.000, E1   +71.154, E3 +48643.777}
SPL {X  -141.358, Y  +310.748, Z    +0.000, E1   +71.233, E3 +48656.482}
SPL {X  -134.330, Y  +298.778, Z    +0.000, E1   +70.323, E3 +48670.330}
SPL {X  -128.957, Y  +290.989, Z    +0.000, E1   +69.528, E3 +48679.695}
SPL {X  -124.846, Y  +285.632, Z    +0.000, E1   +68.906, E3 +48686.158}
SPL {X  -121.783, Y  +281.927, Z    +0.000, E1   +68.403, E3 +48690.590}
SPL {X   -79.219, Y  +246.688, Z    +0.000, E1   +55.887, E3 +48812.097}
ENDSPLINE

SPLINE
SPL {X  -125.038, Y  +285.873, Z    +0.000, E1   +53.023, E3 +48989.138}
SPL {X  -149.949, Y  +329.886, Z    +0.000, E1   +41.515, E3 +49010.703}
SPL {X  -157.246, Y  +356.141, Z    +0.000, E1   +27.282, E3 +49015.760}
SPL {X  -159.525, Y  +373.376, Z    +0.000, E1   +13.812, E3 +49017.417}
SPL {X  -160.000, Y  +387.264, Z    +0.000, E1    +0.544, E3 +49017.874}
SPL {X  -160.000, Y  +390.384, Z    +0.000, E1    -6.008, E3 +49017.912}
SPL {X  -160.000, Y  +395.752, Z    +0.000, E1   -19.038, E3 +49018.105}
SPL {X  -160.000, Y  +404.289, Z    +0.000, E1   -38.292, E3 +49018.774}
SPL {X  -160.000, Y  +418.681, Z    +0.000, E1   -56.949, E3 +49020.963}
SPL {X  -160.000, Y  +471.977, Z    +0.000, E1   -70.792, E3 +49037.483}
SPL {X  -159.977, Y  +677.138, Z    +0.000, E1   -73.665, E3 +49133.974}
SPL {X  -157.805, Y  +700.810, Z    +0.000, E1   -73.511, E3 +49150.804}
SPL {X  -152.242, Y  +723.618, Z    +0.000, E1   -72.940, E3 +49170.717}
SPL {X  -145.929, Y  +740.010, Z    +0.000, E1   -72.229, E3 +49187.188}
SPL {X  -139.114, Y  +753.439, Z    +0.000, E1   -71.436, E3 +49201.827}
SPL {X  -132.333, Y  +764.333, Z    +0.000, E1   -70.535, E3 +49214.451}
SPL {X  -125.486, Y  +773.664, Z    +0.000, E1   -69.598, E3 +49225.425}
SPL {X  -121.321, Y  +778.713, Z    +0.000, E1   -68.872, E3 +49231.435}
SPL {X   -77.337, Y  +814.468, Z    +0.000, E1   -56.377, E3 +49350.066}
ENDSPLINE

SPLINE
SPL {X  -134.727, Y  +760.706, Z    +0.000, E1   -50.460, E3 +49538.298}
SPL {X  -155.580, Y  +711.748, Z    +0.000, E1   -32.084, E3 +49555.213}
SPL {X  -159.445, Y  +687.715, Z    +0.000, E1   -14.660, E3 +49558.059}
SPL {X  -159.995, Y  +675.725, Z    +0.000, E1    -3.424, E3 +49558.570}
SPL {X  -160.000, Y  +671.714, Z    +0.000, E1    +0.835, E3 +49558.611}
SPL {X  -160.000, Y  +663.084, Z    +0.000, E1   +21.134, E3 +49558.935}
SPL {X  -160.000, Y  +650.910, Z    +0.000, E1   +46.005, E3 +49560.089}
SPL {X  -160.000, Y  +634.843, Z    +0.000, E1   +61.273, E3 +49562.766}
SPL {X  -160.000, Y  +578.679, Z    +0.000, E1   +71.665, E3 +49580.599}
SPL {X  -160.000, Y  +387.528, Z    +0.000, E1   +73.487, E3 +49673.412}
SPL {X  -159.218, Y  +369.903, Z    +0.000, E1   +73.425, E3 +49685.279}
SPL {X  -156.808, Y  +353.900, Z    +0.000, E1   +73.180, E3 +49697.883}
SPL {X  -154.539, Y  +344.254, Z    +0.000, E1   +72.827, E3 +49707.420}
ENDSPLINE

SPLINE
SPL {X  -157.258, Y  +356.206, Z    +0.000, E1   +70.434, E3 +49721.992}
ENDSPLINE

SPLINE
SPL {X  -150.342, Y  +330.952, Z    +0.000, E1   +71.154, E3 +49733.665}
SPL {X  -141.358, Y  +310.748, Z    +0.000, E1   +71.233, E3 +49746.370}
SPL {X  -134.330, Y  +298.778, Z    +0.000, E1   +70.323, E3 +49760.218}
SPL {X  -128.957, Y  +290.989, Z    +0.000, E1   +69.528, E3 +49769.583}
SPL {X  -124.846, Y  +285.632, Z    +0.000, E1   +68.906, E3 +49776.046}
SPL {X  -121.783, Y  +281.927, Z    +0.000, E1   +68.403, E3 +49780.478}
SPL {X   -79.219, Y  +246.688, Z    +0.000, E1   +55.887, E3 +49901.985}
ENDSPLINE

SPLINE
SPL {X  -125.038, Y  +285.873, Z    +0.000, E1   +53.023, E3 +50079.026}
SPL {X  -149.949, Y  +329.886, Z    +0.000, E1   +41.515, E3 +50100.591}
SPL {X  -157.246, Y  +356.141, Z    +0.000, E1   +27.282, E3 +50105.648}
SPL {X  -159.525, Y  +373.376, Z    +0.000, E1   +13.812, E3 +50107.305}
SPL {X  -160.000, Y  +387.264, Z    +0.000, E1    +0.544, E3 +50107.762}
SPL {X  -160.000, Y  +390.384, Z    +0.000, E1    -6.008, E3 +50107.800}
SPL {X  -160.000, Y  +395.752, Z    +0.000, E1   -19.038, E3 +50107.993}
SPL {X  -160.000, Y  +404.289, Z    +0.000, E1   -38.292, E3 +50108.662}
SPL {X  -160.000, Y  +418.681, Z    +0.000, E1   -56.949, E3 +50110.851}
SPL {X  -160.000, Y  +471.977, Z    +0.000, E1   -70.792, E3 +50127.371}
SPL {X  -159.977, Y  +677.138, Z    +0.000, E1   -73.665, E3 +50223.862}
SPL {X  -157.805, Y  +700.810, Z    +0.000, E1   -73.511, E3 +50240.692}
SPL {X  -152.242, Y  +723.618, Z    +0.000, E1   -72.940, E3 +50260.605}
SPL {X  -145.929, Y  +740.010, Z    +0.000, E1   -72.229, E3 +50277.076}
SPL {X  -139.114, Y  +753.439, Z    +0.000, E1   -71.436, E3 +50291.715}
SPL {X  -132.333, Y  +764.333, Z    +0.000, E1   -70.535, E3 +50304.339}
SPL {X  -125.486, Y  +773.664, Z    +0.000, E1   -69.598, E3 +50315.313}
SPL {X  -121.321, Y  +778.713, Z    +0.000, E1   -68.872, E3 +50321.323}
SPL {X   -77.337, Y  +814.468, Z    +0.000, E1   -56.377, E3 +50439.954}
ENDSPLINE

SPLINE
SPL {X  -134.727, Y  +760.706, Z    +0.000, E1   -50.460, E3 +50628.186}
SPL {X  -155.580, Y  +711.748, Z    +0.000, E1   -32.084, E3 +50645.101}
SPL {X  -159.445, Y  +687.715, Z    +0.000, E1   -14.660, E3 +50647.947}
SPL {X  -159.995, Y  +675.725, Z    +0.000, E1    -3.424, E3 +50648.458}
SPL {X  -160.000, Y  +671.714, Z    +0.000, E1    +0.835, E3 +50648.499}
SPL {X  -160.000, Y  +663.084, Z    +0.000, E1   +21.134, E3 +50648.823}
SPL {X  -160.000, Y  +650.910, Z    +0.000, E1   +46.005, E3 +50649.977}
SPL {X  -160.000, Y  +634.843, Z    +0.000, E1   +61.273, E3 +50652.654}
SPL {X  -160.000, Y  +578.679, Z    +0.000, E1   +71.665, E3 +50670.487}
SPL {X  -160.000, Y  +387.528, Z    +0.000, E1   +73.487, E3 +50763.300}
SPL {X  -159.218, Y  +369.903, Z    +0.000, E1   +73.425, E3 +50775.167}
SPL {X  -156.808, Y  +353.900, Z    +0.000, E1   +73.180, E3 +50787.771}
SPL {X  -154.539, Y  +344.254, Z    +0.000, E1   +72.827, E3 +50797.308}
ENDSPLINE

SPLINE
SPL {X  -157.258, Y  +356.206, Z    +0.000, E1   +70.434, E3 +50811.880}
ENDSPLINE

SPLINE
SPL {X  -150.342, Y  +330.952, Z    +0.000, E1   +71.154, E3 +50823.553}
SPL {X  -141.358, Y  +310.748, Z    +0.000, E1   +71.233, E3 +50836.258}
SPL {X  -134.330, Y  +298.778, Z    +0.000, E1   +70.323, E3 +50850.106}
SPL {X  -128.957, Y  +290.989, Z    +0.000, E1   +69.528, E3 +50859.471}
SPL {X  -124.846, Y  +285.632, Z    +0.000, E1   +68.906, E3 +50865.934}
SPL {X  -121.783, Y  +281.927, Z    +0.000, E1   +68.403, E3 +50870.366}
SPL {X   -79.219, Y  +246.688, Z    +0.000, E1   +55.887, E3 +50991.873}
ENDSPLINE

SPLINE
SPL {X  -125.038, Y  +285.873, Z    +0.000, E1   +53.023, E3 +51168.914}
SPL {X  -149.949, Y  +329.886, Z    +0.000, E1   +41.515, E3 +51190.479}
SPL {X  -157.246, Y  +356.141, Z    +0.000, E1   +27.282, E3 +51195.536}
SPL {X  -159.525, Y  +373.376, Z    +0.000, E1   +13.812, E3 +51197.193}
SPL {X  -160.000, Y  +387.264, Z    +0.000, E1    +0.544, E3 +51197.650}
SPL {X  -160.000, Y  +390.384, Z    +0.000, E1    -6.008, E3 +51197.688}
SPL {X  -160.000, Y  +395.752, Z    +0.000, E1   -19.038, E3 +51197.881}
SPL {X  -160.000, Y  +404.289, Z    +0.000, E1   -38.292, E3 +51198.550}
SPL {X  -160.000, Y  +418.681, Z    +0.000, E1   -56.949, E3 +51200.739}
SPL {X  -160.000, Y  +471.977, Z    +0.000, E1   -70.792, E3 +51217.259}
SPL {X  -159.977, Y  +677.138, Z    +0.000, E1   -73.665, E3 +51313.750}
SPL {X  -157.805, Y  +700.810, Z    +0.000, E1   -73.511, E3 +51330.580}
SPL {X  -152.242, Y  +723.618, Z    +0.000, E1   -72.940, E3 +51350.493}
SPL {X  -145.929, Y  +740.010, Z    +0.000, E1   -72.229, E3 +51366.964}
SPL {X  -139.114, Y  +753.439, Z    +0.000, E1   -71.436, E3 +51381.603}
SPL {X  -132.333, Y  +764.333, Z    +0.000, E1   -70.535, E3 +51394.227}
SPL {X  -125.486, Y  +773.664, Z    +0.000, E1   -69.598, E3 +51405.201}
SPL {X  -121.321, Y  +778.713, Z    +0.000, E1   -68.872, E3 +51411.211}
SPL {X   -77.337, Y  +814.468, Z    +0.000, E1   -56.377, E3 +51529.842}
ENDSPLINE

SPLINE
SPL {X  -134.727, Y  +760.706, Z    +0.000, E1   -50.460, E3 +51718.074}
SPL {X  -155.580, Y  +711.748, Z    +0.000, E1   -32.084, E3 +51734.989}
SPL {X  -159.445, Y  +687.715, Z    +0.000, E1   -14.660, E3 +51737.835}
SPL {X  -159.995, Y  +675.725, Z    +0.000, E1    -3.424, E3 +51738.346}
SPL {X  -160.000, Y  +671.714, Z    +0.000, E1    +0.835, E3 +51738.387}
SPL {X  -160.000, Y  +663.084, Z    +0.000, E1   +21.134, E3 +51738.711}
SPL {X  -160.000, Y  +650.910, Z    +0.000, E1   +46.005, E3 +51739.865}
SPL {X  -160.000, Y  +634.843, Z    +0.000, E1   +61.273, E3 +51742.542}
SPL {X  -160.000, Y  +578.679, Z    +0.000, E1   +71.665, E3 +51760.375}
SPL {X  -160.000, Y  +387.528, Z    +0.000, E1   +73.487, E3 +51853.188}
SPL {X  -159.218, Y  +369.903, Z    +0.000, E1   +73.425, E3 +51865.055}
SPL {X  -156.808, Y  +353.900, Z    +0.000, E1   +73.180, E3 +51877.659}
SPL {X  -154.539, Y  +344.254, Z    +0.000, E1   +72.827, E3 +51887.196}
ENDSPLINE

SPLINE
SPL {X  -157.258, Y  +356.206, Z    +0.000, E1   +70.434, E3 +51901.768}
ENDSPLINE

SPLINE
SPL {X  -150.342, Y  +330.952, Z    +0.000, E1   +71.154, E3 +51913.441}
SPL {X  -141.358, Y  +310.748, Z    +0.000, E1   +71.233, E3 +51926.147}
SPL {X  -134.330, Y  +298.778, Z    +0.000, E1   +70.323, E3 +51939.994}
SPL {X  -128.957, Y  +290.989, Z    +0.000, E1   +69.528, E3 +51949.359}
SPL {X  -124.846, Y  +285.632, Z    +0.000, E1   +68.906, E3 +51955.822}
SPL {X  -121.783, Y  +281.927, Z    +0.000, E1   +68.403, E3 +51960.255}
SPL {X   -79.219, Y  +246.688, Z    +0.000, E1   +55.887, E3 +52081.761}
ENDSPLINE

SPLINE
SPL {X  -125.038, Y  +285.873, Z    +0.000, E1   +53.023, E3 +52258.802}
SPL {X  -149.949, Y  +329.886, Z    +0.000, E1   +41.515, E3 +52280.367}
SPL {X  -157.246, Y  +356.141, Z    +0.000, E1   +27.282, E3 +52285.424}
SPL {X  -159.525, Y  +373.376, Z    +0.000, E1   +13.812, E3 +52287.081}
SPL {X  -160.000, Y  +387.264, Z    +0.000, E1    +0.544, E3 +52287.538}
SPL {X  -160.000, Y  +390.384, Z    +0.000, E1    -6.008, E3 +52287.576}
SPL {X  -160.000, Y  +395.752, Z    +0.000, E1   -19.038, E3 +52287.769}
SPL {X  -160.000, Y  +404.289, Z    +0.000, E1   -38.292, E3 +52288.438}
SPL {X  -160.000, Y  +418.681, Z    +0.000, E1   -56.949, E3 +52290.627}
SPL {X  -160.000, Y  +471.977, Z    +0.000, E1   -70.792, E3 +52307.147}
SPL {X  -159.977, Y  +677.138, Z    +0.000, E1   -73.665, E3 +52403.638}
SPL {X  -157.805, Y  +700.810, Z    +0.000, E1   -73.511, E3 +52420.468}
SPL {X  -152.242, Y  +723.618, Z    +0.000, E1   -72.940, E3 +52440.381}
SPL {X  -145.929, Y  +740.010, Z    +0.000, E1   -72.229, E3 +52456.852}
SPL {X  -139.114, Y  +753.439, Z    +0.000, E1   -71.436, E3 +52471.491}
SPL {X  -132.333, Y  +764.333, Z    +0.000, E1   -70.535, E3 +52484.115}
SPL {X  -125.486, Y  +773.664, Z    +0.000, E1   -69.598, E3 +52495.089}
SPL {X  -121.321, Y  +778.713, Z    +0.000, E1   -68.872, E3 +52501.099}
SPL {X   -77.337, Y  +814.468, Z    +0.000, E1   -56.377, E3 +52619.730}
ENDSPLINE

SPLINE
SPL {X  -134.727, Y  +760.706, Z    +0.000, E1   -50.460, E3 +52807.962}
SPL {X  -155.580, Y  +711.748, Z    +0.000, E1   -32.084, E3 +52824.877}
SPL {X  -159.445, Y  +687.715, Z    +0.000, E1   -14.660, E3 +52827.724}
SPL {X  -159.995, Y  +675.725, Z    +0.000, E1    -3.424, E3 +52828.234}
SPL {X  -160.000, Y  +671.714, Z    +0.000, E1    +0.835, E3 +52828.275}
SPL {X  -160.000, Y  +663.084, Z    +0.000, E1   +21.134, E3 +52828.599}
SPL {X  -160.000, Y  +650.910, Z    +0.000, E1   +46.005, E3 +52829.753}
SPL {X  -160.000, Y  +634.843, Z    +0.000, E1   +61.273, E3 +52832.430}
SPL {X  -160.000, Y  +578.679, Z    +0.000, E1   +71.665, E3 +52850.263}
SPL {X  -160.000, Y  +387.528, Z    +0.000, E1   +73.487, E3 +52943.076}
SPL {X  -159.218, Y  +369.903, Z    +0.000, E1   +73.425, E3 +52954.943}
SPL {X  -156.808, Y  +353.900, Z    +0.000, E1   +73.180, E3 +52967.547}
SPL {X  -154.539, Y  +344.254, Z    +0.000, E1   +72.827, E3 +52977.084}
ENDSPLINE

SPLINE
SPL {X  -157.258, Y  +356.206, Z    +0.000, E1   +70.434, E3 +52991.657}
ENDSPLINE

SPLINE
SPL {X  -150.342, Y  +330.952, Z    +0.000, E1   +71.154, E3 +53003.329}
SPL {X  -141.358, Y  +310.748, Z    +0.000, E1   +71.233, E3 +53016.035}
SPL {X  -134.330, Y  +298.778, Z    +0.000, E1   +70.323, E3 +53029.882}
SPL {X  -128.957, Y  +290.989, Z    +0.000, E1   +69.528, E3 +53039.247}
SPL {X  -124.846, Y  +285.632, Z    +0.000, E1   +68.906, E3 +53045.710}
SPL {X  -121.783, Y  +281.927, Z    +0.000, E1   +68.403, E3 +53050.143}
SPL {X   -79.219, Y  +246.688, Z    +0.000, E1   +55.887, E3 +53171.649}
ENDSPLINE

SPLINE
SPL {X  -125.038, Y  +285.873, Z    +0.000, E1   +53.023, E3 +53348.690}
SPL {X  -149.949, Y  +329.886, Z    +0.000, E1   +41.515, E3 +53370.255}
SPL {X  -157.246, Y  +356.141, Z    +0.000, E1   +27.282, E3 +53375.312}
SPL {X  -159.525, Y  +373.376, Z    +0.000, E1   +13.812, E3 +53376.969}
SPL {X  -160.000, Y  +387.264, Z    +0.000, E1    +0.544, E3 +53377.426}
SPL {X  -160.000, Y  +390.384, Z    +0.000, E1    -6.008, E3 +53377.464}
SPL {X  -160.000, Y  +395.752, Z    +0.000, E1   -19.038, E3 +53377.657}
SPL {X  -160.000, Y  +404.289, Z    +0.000, E1   -38.292, E3 +53378.326}
SPL {X  -160.000, Y  +418.681, Z    +0.000, E1   -56.949, E3 +53380.515}
SPL {X  -160.000, Y  +471.977, Z    +0.000, E1   -70.792, E3 +53397.035}
SPL {X  -159.977, Y  +677.138, Z    +0.000, E1   -73.665, E3 +53493.526}
SPL {X  -157.805, Y  +700.810, Z    +0.000, E1   -73.511, E3 +53510.356}
SPL {X  -152.242, Y  +723.618, Z    +0.000, E1   -72.940, E3 +53530.269}
SPL {X  -145.929, Y  +740.010, Z    +0.000, E1   -72.229, E3 +53546.740}
SPL {X  -139.114, Y  +753.439, Z    +0.000, E1   -71.436, E3 +53561.379}
SPL {X  -132.333, Y  +764.333, Z    +0.000, E1   -70.535, E3 +53574.003}
SPL {X  -125.486, Y  +773.664, Z    +0.000, E1   -69.598, E3 +53584.977}
SPL {X  -121.321, Y  +778.713, Z    +0.000, E1   -68.872, E3 +53590.987}
SPL {X   -77.337, Y  +814.468, Z    +0.000, E1   -56.377, E3 +53709.618}
ENDSPLINE

SPLINE
SPL {X  -134.727, Y  +760.706, Z    +0.000, E1   -50.460, E3 +53897.850}
SPL {X  -155.580, Y  +711.748, Z    +0.000, E1   -32.084, E3 +53914.765}
SPL {X  -159.445, Y  +687.715, Z    +0.000, E1   -14.660, E3 +53917.612}
SPL {X  -159.995, Y  +675.725, Z    +0.000, E1    -3.424, E3 +53918.122}
SPL {X  -160.000, Y  +671.714, Z    +0.000, E1    +0.835, E3 +53918.163}
SPL {X  -160.000, Y  +663.084, Z    +0.000, E1   +21.134, E3 +53918.487}
SPL {X  -160.000, Y  +650.910, Z    +0.000, E1   +46.005, E3 +53919.641}
SPL {X  -160.000, Y  +634.843, Z    +0.000, E1   +61.273, E3 +53922.318}
SPL {X  -160.000, Y  +578.679, Z    +0.000, E1   +71.665, E3 +53940.151}
SPL {X  -160.000, Y  +387.528, Z    +0.000, E1   +73.487, E3 +54032.964}
SPL {X  -159.218, Y  +369.903, Z    +0.000, E1   +73.425, E3 +54044.831}
SPL {X  -156.808, Y  +353.900, Z    +0.000, E1   +73.180, E3 +54057.435}
SPL {X  -154.539, Y  +344.254, Z    +0.000, E1   +72.827, E3 +54066.972}
ENDSPLINE

SPLINE
SPL {X  -157.258, Y  +356.206, Z    +0.000, E1   +70.434, E3 +54081.545}
ENDSPLINE

SPLINE
SPL {X  -150.342, Y  +330.952, Z    +0.000, E1   +71.154, E3 +54093.217}
SPL {X  -141.358, Y  +310.748, Z    +0.000, E1   +71.233, E3 +54105.923}
SPL {X  -134.330, Y  +298.778, Z    +0.000, E1   +70.323, E3 +54119.770}
SPL {X  -128.957, Y  +290.989, Z    +0.000, E1   +69.528, E3 +54129.135}
SPL {X  -124.846, Y  +285.632, Z    +0.000, E1   +68.906, E3 +54135.598}
SPL {X  -121.783, Y  +281.927, Z    +0.000, E1   +68.403, E3 +54140.031}
SPL {X   -79.219, Y  +246.688, Z    +0.000, E1   +55.887, E3 +54261.537}
ENDSPLINE

SPLINE
SPL {X  -125.038, Y  +285.873, Z    +0.000, E1   +53.023, E3 +54438.578}
SPL {X  -149.949, Y  +329.886, Z    +0.000, E1   +41.515, E3 +54460.143}
SPL {X  -157.246, Y  +356.141, Z    +0.000, E1   +27.282, E3 +54465.200}
SPL {X  -159.525, Y  +373.376, Z    +0.000, E1   +13.812, E3 +54466.857}
SPL {X  -160.000, Y  +387.264, Z    +0.000, E1    +0.544, E3 +54467.315}
SPL {X  -160.000, Y  +390.384, Z    +0.000, E1    -6.008, E3 +54467.352}
SPL {X  -160.000, Y  +395.752, Z    +0.000, E1   -19.038, E3 +54467.545}
SPL {X  -160.000, Y  +404.289, Z    +0.000, E1   -38.292, E3 +54468.214}
SPL {X  -160.000, Y  +418.681, Z    +0.000, E1   -56.949, E3 +54470.404}
SPL {X  -160.000, Y  +471.977, Z    +0.000, E1   -70.792, E3 +54486.923}
SPL {X  -159.977, Y  +677.138, Z    +0.000, E1   -73.665, E3 +54583.414}
SPL {X  -157.805, Y  +700.810, Z    +0.000, E1   -73.511, E3 +54600.244}
SPL {X  -152.242, Y  +723.618, Z    +0.000, E1   -72.940, E3 +54620.157}
SPL {X  -145.929, Y  +740.010, Z    +0.000, E1   -72.229, E3 +54636.628}
SPL {X  -139.114, Y  +753.439, Z    +0.000, E1   -71.436, E3 +54651.267}
SPL {X  -132.333, Y  +764.333, Z    +0.000, E1   -70.535, E3 +54663.891}
SPL {X  -125.486, Y  +773.664, Z    +0.000, E1   -69.598, E3 +54674.865}
SPL {X  -121.321, Y  +778.713, Z    +0.000, E1   -68.872, E3 +54680.875}
SPL {X   -77.337, Y  +814.468, Z    +0.000, E1   -56.377, E3 +54799.506}
ENDSPLINE

SPLINE
SPL {X  -134.727, Y  +760.706, Z    +0.000, E1   -50.460, E3 +54987.738}
SPL {X  -155.580, Y  +711.748, Z    +0.000, E1   -32.084, E3 +55004.653}
SPL {X  -159.445, Y  +687.715, Z    +0.000, E1   -14.660, E3 +55007.500}
SPL {X  -159.995, Y  +675.725, Z    +0.000, E1    -3.424, E3 +55008.010}
SPL {X  -160.000, Y  +671.714, Z    +0.000, E1    +0.835, E3 +55008.051}
SPL {X  -160.000, Y  +663.084, Z    +0.000, E1   +21.134, E3 +55008.375}
SPL {X  -160.000, Y  +650.910, Z    +0.000, E1   +46.005, E3 +55009.529}
SPL {X  -160.000, Y  +634.843, Z    +0.000, E1   +61.273, E3 +55012.206}
SPL {X  -160.000, Y  +578.679, Z    +0.000, E1   +71.665, E3 +55030.039}
SPL {X  -160.000, Y  +387.528, Z    +0.000, E1   +73.487, E3 +55122.852}
SPL {X  -159.218, Y  +369.903, Z    +0.000, E1   +73.425, E3 +55134.719}
SPL {X  -156.808, Y  +353.900, Z    +0.000, E1   +73.180, E3 +55147.323}
SPL {X  -154.539, Y  +344.254, Z    +0.000, E1   +72.827, E3 +55156.860}
ENDSPLINE

SPLINE
SPL {X  -157.258, Y  +356.206, Z    +0.000, E1   +70.434, E3 +55171.433}
ENDSPLINE

SPLINE
SPL {X  -150.342, Y  +330.952, Z    +0.000, E1   +71.154, E3 +55183.105}
SPL {X  -141.358, Y  +310.748, Z    +0.000, E1   +71.233, E3 +55195.811}
SPL {X  -134.330, Y  +298.778, Z    +0.000, E1   +70.323, E3 +55209.658}
SPL {X  -128.957, Y  +290.989, Z    +0.000, E1   +69.528, E3 +55219.023}
SPL {X  -124.846, Y  +285.632, Z    +0.000, E1   +68.906, E3 +55225.486}
SPL {X  -121.783, Y  +281.927, Z    +0.000, E1   +68.403, E3 +55229.919}
SPL {X   -79.219, Y  +246.688, Z    +0.000, E1   +55.887, E3 +55351.425}
ENDSPLINE

SPLINE
SPL {X  -125.038, Y  +285.873, Z    +0.000, E1   +53.023, E3 +55528.466}
SPL {X  -149.949, Y  +329.886, Z    +0.000, E1   +41.515, E3 +55550.031}
SPL {X  -157.246, Y  +356.141, Z    +0.000, E1   +27.282, E3 +55555.088}
SPL {X  -159.525, Y  +373.376, Z    +0.000, E1   +13.812, E3 +55556.745}
SPL {X  -160.000, Y  +387.264, Z    +0.000, E1    +0.544, E3 +55557.203}
SPL {X  -160.000, Y  +390.384, Z    +0.000, E1    -6.008, E3 +55557.240}
SPL {X  -160.000, Y  +395.752, Z    +0.000, E1   -19.038, E3 +55557.433}
SPL {X  -160.000, Y  +404.289, Z    +0.000, E1   -38.292, E3 +55558.102}
SPL {X  -160.000, Y  +418.681, Z    +0.000, E1   -56.949, E3 +55560.292}
SPL {X  -160.000, Y  +471.977, Z    +0.000, E1   -70.792, E3 +55576.811}
SPL {X  -159.977, Y  +677.138, Z    +0.000, E1   -73.665, E3 +55673.302}
SPL {X  -157.805, Y  +700.810, Z    +0.000, E1   -73.511, E3 +55690.132}
SPL {X  -152.242, Y  +723.618, Z    +0.000, E1   -72.940, E3 +55710.045}
SPL {X  -145.929, Y  +740.010, Z    +0.000, E1   -72.229, E3 +55726.516}
SPL {X  -139.114, Y  +753.439, Z    +0.000, E1   -71.436, E3 +55741.155}
SPL {X  -132.333, Y  +764.333, Z    +0.000, E1   -70.535, E3 +55753.779}
SPL {X  -125.486, Y  +773.664, Z    +0.000, E1   -69.598, E3 +55764.753}
SPL {X  -121.321, Y  +778.713, Z    +0.000, E1   -68.872, E3 +55770.763}
SPL {X   -77.337, Y  +814.468, Z    +0.000, E1   -56.377, E3 +55889.394}
ENDSPLINE

SPLINE
SPL {X  -134.727, Y  +760.706, Z    +0.000, E1   -50.460, E3 +56077.626}
SPL {X  -155.580, Y  +711.748, Z    +0.000, E1   -32.084, E3 +56094.541}
SPL {X  -159.445, Y  +687.715, Z    +0.000, E1   -14.660, E3 +56097.388}
SPL {X  -159.995, Y  +675.725, Z    +0.000, E1    -3.424, E3 +56097.898}
SPL {X  -160.000, Y  +671.714, Z    +0.000, E1    +0.835, E3 +56097.939}
SPL {X  -160.000, Y  +663.084, Z    +0.000, E1   +21.134, E3 +56098.263}
SPL {X  -160.000, Y  +650.910, Z    +0.000, E1   +46.005, E3 +56099.417}
SPL {X  -160.000, Y  +634.843, Z    +0.000, E1   +61.273, E3 +56102.094}
SPL {X  -160.000, Y  +578.679, Z    +0.000, E1   +71.665, E3 +56119.927}
SPL {X  -160.000, Y  +387.528, Z    +0.000, E1   +73.487, E3 +56212.740}
SPL {X  -159.218, Y  +369.903, Z    +0.000, E1   +73.425, E3 +56224.607}
SPL {X  -156.808, Y  +353.900, Z    +0.000, E1   +73.180, E3 +56237.211}
SPL {X  -154.539, Y  +344.254, Z    +0.000, E1   +72.827, E3 +56246.748}
ENDSPLINE

SPLINE
SPL {X  -157.258, Y  +356.206, Z    +0.000, E1   +70.434, E3 +56261.321}
ENDSPLINE

SPLINE
SPL {X  -150.342, Y  +330.952, Z    +0.000, E1   +71.154, E3 +56272.993}
SPL {X  -141.358, Y  +310.748, Z    +0.000, E1   +71.233, E3 +56285.699}
SPL {X  -134.330, Y  +298.778, Z    +0.000, E1   +70.323, E3 +56299.546}
SPL {X  -128.957, Y  +290.989, Z    +0.000, E1   +69.528, E3 +56308.911}
SPL {X  -124.846, Y  +285.632, Z    +0.000, E1   +68.906, E3 +56315.374}
SPL {X  -121.783, Y  +281.927, Z    +0.000, E1   +68.403, E3 +56319.807}
SPL {X   -79.219, Y  +246.688, Z    +0.000, E1   +55.887, E3 +56441.313}
ENDSPLINE

SPLINE
SPL {X  -125.038, Y  +285.873, Z    +0.000, E1   +53.023, E3 +56618.354}
SPL {X  -149.949, Y  +329.886, Z    +0.000, E1   +41.515, E3 +56639.919}
SPL {X  -157.246, Y  +356.141, Z    +0.000, E1   +27.282, E3 +56644.976}
SPL {X  -159.525, Y  +373.376, Z    +0.000, E1   +13.812, E3 +56646.633}
SPL {X  -160.000, Y  +387.264, Z    +0.000, E1    +0.544, E3 +56647.091}
SPL {X  -160.000, Y  +390.384, Z    +0.000, E1    -6.008, E3 +56647.128}
SPL {X  -160.000, Y  +395.752, Z    +0.000, E1   -19.038, E3 +56647.321}
SPL {X  -160.000, Y  +404.289, Z    +0.000, E1   -38.292, E3 +56647.990}
SPL {X  -160.000, Y  +418.681, Z    +0.000, E1   -56.949, E3 +56650.180}
SPL {X  -160.000, Y  +471.977, Z    +0.000, E1   -70.792, E3 +56666.699}
SPL {X  -159.977, Y  +677.138, Z    +0.000, E1   -73.665, E3 +56763.190}
SPL {X  -157.805, Y  +700.810, Z    +0.000, E1   -73.511, E3 +56780.020}
SPL {X  -152.242, Y  +723.618, Z    +0.000, E1   -72.940, E3 +56799.933}
SPL {X  -145.929, Y  +740.010, Z    +0.000, E1   -72.229, E3 +56816.404}
SPL {X  -139.114, Y  +753.439, Z    +0.000, E1   -71.436, E3 +56831.043}
SPL {X  -132.333, Y  +764.333, Z    +0.000, E1   -70.535, E3 +56843.667}
SPL {X  -125.486, Y  +773.664, Z    +0.000, E1   -69.598, E3 +56854.641}
SPL {X  -121.321, Y  +778.713, Z    +0.000, E1   -68.872, E3 +56860.651}
SPL {X   -77.337, Y  +814.468, Z    +0.000, E1   -56.377, E3 +56979.282}
ENDSPLINE

SPLINE
SPL {X  -134.727, Y  +760.706, Z    +0.000, E1   -50.460, E3 +57167.514}
SPL {X  -155.580, Y  +711.748, Z    +0.000, E1   -32.084, E3 +57184.429}
SPL {X  -159.445, Y  +687.715, Z    +0.000, E1   -14.660, E3 +57187.276}
SPL {X  -159.995, Y  +675.725, Z    +0.000, E1    -3.424, E3 +57187.786}
SPL {X  -160.000, Y  +671.714, Z    +0.000, E1    +0.835, E3 +57187.827}
SPL {X  -160.000, Y  +663.084, Z    +0.000, E1   +21.134, E3 +57188.151}
SPL {X  -160.000, Y  +650.910, Z    +0.000, E1   +46.005, E3 +57189.305}
SPL {X  -160.000, Y  +634.843, Z    +0.000, E1   +61.273, E3 +57191.982}
SPL {X  -160.000, Y  +578.679, Z    +0.000, E1   +71.665, E3 +57209.816}
SPL {X  -160.000, Y  +387.528, Z    +0.000, E1   +73.487, E3 +57302.628}
SPL {X  -159.218, Y  +369.903, Z    +0.000, E1   +73.425, E3 +57314.495}
SPL {X  -156.808, Y  +353.900, Z    +0.000, E1   +73.180, E3 +57327.099}
SPL {X  -154.539, Y  +344.254, Z    +0.000, E1   +72.827, E3 +57336.636}
ENDSPLINE

SPLINE
SPL {X  -157.258, Y  +356.206, Z    +0.000, E1   +70.434, E3 +57351.209}
ENDSPLINE

SPLINE
SPL {X  -150.342, Y  +330.952, Z    +0.000, E1   +71.154, E3 +57362.881}
SPL {X  -141.358, Y  +310.748, Z    +0.000, E1   +71.233, E3 +57375.587}
SPL {X  -134.330, Y  +298.778, Z    +0.000, E1   +70.323, E3 +57389.434}
SPL {X  -128.957, Y  +290.989, Z    +0.000, E1   +69.528, E3 +57398.799}
SPL {X  -124.846, Y  +285.632, Z    +0.000, E1   +68.906, E3 +57405.262}
SPL {X  -121.783, Y  +281.927, Z    +0.000, E1   +68.403, E3 +57409.695}
SPL {X   -79.219, Y  +246.688, Z    +0.000, E1   +55.887, E3 +57531.201}
ENDSPLINE

SPLINE
SPL {X  -125.038, Y  +285.873, Z    +0.000, E1   +53.023, E3 +57708.242}
SPL {X  -149.949, Y  +329.886, Z    +0.000, E1   +41.515, E3 +57729.807}
SPL {X  -157.246, Y  +356.141, Z    +0.000, E1   +27.282, E3 +57734.864}
SPL {X  -159.525, Y  +373.376, Z    +0.000, E1   +13.812, E3 +57736.521}
SPL {X  -160.000, Y  +387.264, Z    +0.000, E1    +0.544, E3 +57736.979}
SPL {X  -160.000, Y  +390.384, Z    +0.000, E1    -6.008, E3 +57737.016}
SPL {X  -160.000, Y  +395.752, Z    +0.000, E1   -19.038, E3 +57737.209}
SPL {X  -160.000, Y  +404.289, Z    +0.000, E1   -38.292, E3 +57737.878}
SPL {X  -160.000, Y  +418.681, Z    +0.000, E1   -56.949, E3 +57740.068}
SPL {X  -160.000, Y  +471.977, Z    +0.000, E1   -70.792, E3 +57756.587}
SPL {X  -159.977, Y  +677.138, Z    +0.000, E1   -73.665, E3 +57853.078}
SPL {X  -157.805, Y  +700.810, Z    +0.000, E1   -73.511, E3 +57869.908}
SPL {X  -152.242, Y  +723.618, Z    +0.000, E1   -72.940, E3 +57889.821}
SPL {X  -145.929, Y  +740.010, Z    +0.000, E1   -72.229, E3 +57906.292}
SPL {X  -139.114, Y  +753.439, Z    +0.000, E1   -71.436, E3 +57920.931}
SPL {X  -132.333, Y  +764.333, Z    +0.000, E1   -70.535, E3 +57933.555}
SPL {X  -125.486, Y  +773.664, Z    +0.000, E1   -69.598, E3 +57944.529}
SPL {X  -121.321, Y  +778.713, Z    +0.000, E1   -68.872, E3 +57950.539}
SPL {X   -77.337, Y  +814.468, Z    +0.000, E1   -56.377, E3 +58069.170}
ENDSPLINE

SPLINE
SPL {X  -134.727, Y  +760.706, Z    +0.000, E1   -50.460, E3 +58257.402}
SPL {X  -155.580, Y  +711.748, Z    +0.000, E1   -32.084, E3 +58274.317}
SPL {X  -159.445, Y  +687.715, Z    +0.000, E1   -14.660, E3 +58277.164}
SPL {X  -159.995, Y  +675.725, Z    +0.000, E1    -3.424, E3 +58277.675}
SPL {X  -160.000, Y  +671.714, Z    +0.000, E1    +0.835, E3 +58277.715}
SPL {X  -160.000, Y  +663.084, Z    +0.000, E1   +21.134, E3 +58278.039}
SPL {X  -160.000, Y  +650.910, Z    +0.000, E1   +46.005, E3 +58279.193}
SPL {X  -160.000, Y  +634.843, Z    +0.000, E1   +61.273, E3 +58281.870}
SPL {X  -160.000, Y  +578.679, Z    +0.000, E1   +71.665, E3 +58299.704}
SPL {X  -160.000, Y  +387.528, Z    +0.000, E1   +73.487, E3 +58392.516}
SPL {X  -159.218, Y  +369.903, Z    +0.000, E1   +73.425, E3 +58404.383}
SPL {X  -156.808, Y  +353.900, Z    +0.000, E1   +73.180, E3 +58416.987}
SPL {X  -154.539, Y  +344.254, Z    +0.000, E1   +72.827, E3 +58426.524}
ENDSPLINE

SPLINE
SPL {X  -157.258, Y  +356.206, Z    +0.000, E1   +70.434, E3 +58441.097}
ENDSPLINE

SPLINE
SPL {X  -150.342, Y  +330.952, Z    +0.000, E1   +71.154, E3 +58452.769}
SPL {X  -141.358, Y  +310.748, Z    +0.000, E1   +71.233, E3 +58465.475}
SPL {X  -134.330, Y  +298.778, Z    +0.000, E1   +70.323, E3 +58479.322}
SPL {X  -128.957, Y  +290.989, Z    +0.000, E1   +69.528, E3 +58488.687}
SPL {X  -124.846, Y  +285.632, Z    +0.000, E1   +68.906, E3 +58495.151}
SPL {X  -121.783, Y  +281.927, Z    +0.000, E1   +68.403, E3 +58499.583}
SPL {X   -79.219, Y  +246.688, Z    +0.000, E1   +55.887, E3 +58621.089}
ENDSPLINE

SPLINE
SPL {X  -125.038, Y  +285.873, Z    +0.000, E1   +53.023, E3 +58798.130}
SPL {X  -149.949, Y  +329.886, Z    +0.000, E1   +41.515, E3 +58819.695}
SPL {X  -157.246, Y  +356.141, Z    +0.000, E1   +27.282, E3 +58824.752}
SPL {X  -159.525, Y  +373.376, Z    +0.000, E1   +13.812, E3 +58826.409}
SPL {X  -160.000, Y  +387.264, Z    +0.000, E1    +0.544, E3 +58826.867}
SPL {X  -160.000, Y  +390.384, Z    +0.000, E1    -6.008, E3 +58826.904}
SPL {X  -160.000, Y  +395.752, Z    +0.000, E1   -19.038, E3 +58827.097}
SPL {X  -160.000, Y  +404.289, Z    +0.000, E1   -38.292, E3 +58827.766}
SPL {X  -160.000, Y  +418.681, Z    +0.000, E1   -56.949, E3 +58829.956}
SPL {X  -160.000, Y  +471.977, Z    +0.000, E1   -70.792, E3 +58846.475}
SPL {X  -159.977, Y  +677.138, Z    +0.000, E1   -73.665, E3 +58942.966}
SPL {X  -157.805, Y  +700.810, Z    +0.000, E1   -73.511, E3 +58959.796}
SPL {X  -152.242, Y  +723.618, Z    +0.000, E1   -72.940, E3 +58979.709}
SPL {X  -145.929, Y  +740.010, Z    +0.000, E1   -72.229, E3 +58996.180}
SPL {X  -139.114, Y  +753.439, Z    +0.000, E1   -71.436, E3 +59010.819}
SPL {X  -132.333, Y  +764.333, Z    +0.000, E1   -70.535, E3 +59023.443}
SPL {X  -125.486, Y  +773.664, Z    +0.000, E1   -69.598, E3 +59034.417}
SPL {X  -121.321, Y  +778.713, Z    +0.000, E1   -68.872, E3 +59040.427}
SPL {X   -77.337, Y  +814.468, Z    +0.000, E1   -56.377, E3 +59159.058}
ENDSPLINE

SPLINE
SPL {X  -134.727, Y  +760.706, Z    +0.000, E1   -50.460, E3 +59347.290}
SPL {X  -155.580, Y  +711.748, Z    +0.000, E1   -32.084, E3 +59364.205}
SPL {X  -159.445, Y  +687.715, Z    +0.000, E1   -14.660, E3 +59367.052}
SPL {X  -159.995, Y  +675.725, Z    +0.000, E1    -3.424, E3 +59367.563}
SPL {X  -160.000, Y  +671.714, Z    +0.000, E1    +0.835, E3 +59367.603}
SPL {X  -160.000, Y  +663.084, Z    +0.000, E1   +21.134, E3 +59367.927}
SPL {X  -160.000, Y  +650.910, Z    +0.000, E1   +46.005, E3 +59369.081}
SPL {X  -160.000, Y  +634.843, Z    +0.000, E1   +61.273, E3 +59371.758}
SPL {X  -160.000, Y  +578.679, Z    +0.000, E1   +71.665, E3 +59389.592}
SPL {X  -160.000, Y  +387.528, Z    +0.000, E1   +73.487, E3 +59482.404}
SPL {X  -159.218, Y  +369.903, Z    +0.000, E1   +73.425, E3 +59494.271}
SPL {X  -156.808, Y  +353.900, Z    +0.000, E1   +73.180, E3 +59506.875}
SPL {X  -154.539, Y  +344.254, Z    +0.000, E1   +72.827, E3 +59516.412}
ENDSPLINE

SPLINE
SPL {X  -157.258, Y  +356.206, Z    +0.000, E1   +70.434, E3 +59530.985}
ENDSPLINE

SPLINE
SPL {X  -150.342, Y  +330.952, Z    +0.000, E1   +71.154, E3 +59542.657}
SPL {X  -141.358, Y  +310.748, Z    +0.000, E1   +71.233, E3 +59555.363}
SPL {X  -134.330, Y  +298.778, Z    +0.000, E1   +70.323, E3 +59569.210}
SPL {X  -128.957, Y  +290.989, Z    +0.000, E1   +69.528, E3 +59578.575}
SPL {X  -124.846, Y  +285.632, Z    +0.000, E1   +68.906, E3 +59585.039}
SPL {X  -121.783, Y  +281.927, Z    +0.000, E1   +68.403, E3 +59589.471}
SPL {X   -79.219, Y  +246.688, Z    +0.000, E1   +55.887, E3 +59710.977}
ENDSPLINE

SPLINE
SPL {X  -125.038, Y  +285.873, Z    +0.000, E1   +53.023, E3 +59888.018}
SPL {X  -149.949, Y  +329.886, Z    +0.000, E1   +41.515, E3 +59909.583}
SPL {X  -157.246, Y  +356.141, Z    +0.000, E1   +27.282, E3 +59914.640}
SPL {X  -159.525, Y  +373.376, Z    +0.000, E1   +13.812, E3 +59916.297}
SPL {X  -160.000, Y  +387.264, Z    +0.000, E1    +0.544, E3 +59916.755}
SPL {X  -160.000, Y  +390.384, Z    +0.000, E1    -6.008, E3 +59916.792}
SPL {X  -160.000, Y  +395.752, Z    +0.000, E1   -19.038, E3 +59916.986}
SPL {X  -160.000, Y  +404.289, Z    +0.000, E1   -38.292, E3 +59917.654}
SPL {X  -160.000, Y  +418.681, Z    +0.000, E1   -56.949, E3 +59919.844}
SPL {X  -160.000, Y  +471.977, Z    +0.000, E1   -70.792, E3 +59936.363}
SPL {X  -159.977, Y  +677.138, Z    +0.000, E1   -73.665, E3 +60032.854}
SPL {X  -157.805, Y  +700.810, Z    +0.000, E1   -73.511, E3 +60049.684}
SPL {X  -152.242, Y  +723.618, Z    +0.000, E1   -72.940, E3 +60069.597}
SPL {X  -145.929, Y  +740.010, Z    +0.000, E1   -72.229, E3 +60086.069}
SPL {X  -139.114, Y  +753.439, Z    +0.000, E1   -71.436, E3 +60100.707}
SPL {X  -132.333, Y  +764.333, Z    +0.000, E1   -70.535, E3 +60113.331}
SPL {X  -125.486, Y  +773.664, Z    +0.000, E1   -69.598, E3 +60124.305}
SPL {X  -121.321, Y  +778.713, Z    +0.000, E1   -68.872, E3 +60130.315}
SPL {X   -77.337, Y  +814.468, Z    +0.000, E1   -56.377, E3 +60248.946}
ENDSPLINE

SPLINE
SPL {X  -134.727, Y  +760.706, Z    +0.000, E1   -50.460, E3 +60437.178}
SPL {X  -155.580, Y  +711.748, Z    +0.000, E1   -32.084, E3 +60454.093}
SPL {X  -159.445, Y  +687.715, Z    +0.000, E1   -14.660, E3 +60456.940}
SPL {X  -159.995, Y  +675.725, Z    +0.000, E1    -3.424, E3 +60457.451}
SPL {X  -160.000, Y  +671.714, Z    +0.000, E1    +0.835, E3 +60457.491}
SPL {X  -160.000, Y  +663.084, Z    +0.000, E1   +21.134, E3 +60457.815}
SPL {X  -160.000, Y  +650.910, Z    +0.000, E1   +46.005, E3 +60458.969}
SPL {X  -160.000, Y  +634.843, Z    +0.000, E1   +61.273, E3 +60461.646}
SPL {X  -160.000, Y  +578.679, Z    +0.000, E1   +71.665, E3 +60479.480}
SPL {X  -160.000, Y  +387.528, Z    +0.000, E1   +73.487, E3 +60572.292}
SPL {X  -159.218, Y  +369.903, Z    +0.000, E1   +73.425, E3 +60584.159}
SPL {X  -156.808, Y  +353.900, Z    +0.000, E1   +73.180, E3 +60596.763}
SPL {X  -154.539, Y  +344.254, Z    +0.000, E1   +72.827, E3 +60606.300}
ENDSPLINE

SPLINE
SPL {X  -157.258, Y  +356.206, Z    +0.000, E1   +70.434, E3 +60620.873}
ENDSPLINE

SPLINE
SPL {X  -150.342, Y  +330.952, Z    +0.000, E1   +71.154, E3 +60632.545}
SPL {X  -141.358, Y  +310.748, Z    +0.000, E1   +71.233, E3 +60645.251}
SPL {X  -134.330, Y  +298.778, Z    +0.000, E1   +70.323, E3 +60659.098}
SPL {X  -128.957, Y  +290.989, Z    +0.000, E1   +69.528, E3 +60668.463}
SPL {X  -124.846, Y  +285.632, Z    +0.000, E1   +68.906, E3 +60674.927}
SPL {X  -121.783, Y  +281.927, Z    +0.000, E1   +68.403, E3 +60679.359}
SPL {X   -79.219, Y  +246.688, Z    +0.000, E1   +55.887, E3 +60800.865}
ENDSPLINE

SPLINE
SPL {X  -125.038, Y  +285.873, Z    +0.000, E1   +53.023, E3 +60977.906}
SPL {X  -149.949, Y  +329.886, Z    +0.000, E1   +41.515, E3 +60999.471}
SPL {X  -157.246, Y  +356.141, Z    +0.000, E1   +27.282, E3 +61004.528}
SPL {X  -159.525, Y  +373.376, Z    +0.000, E1   +13.812, E3 +61006.185}
SPL {X  -160.000, Y  +387.264, Z    +0.000, E1    +0.544, E3 +61006.643}
SPL {X  -160.000, Y  +390.384, Z    +0.000, E1    -6.008, E3 +61006.680}
SPL {X  -160.000, Y  +395.752, Z    +0.000, E1   -19.038, E3 +61006.874}
SPL {X  -160.000, Y  +404.289, Z    +0.000, E1   -38.292, E3 +61007.542}
SPL {X  -160.000, Y  +418.681, Z    +0.000, E1   -56.949, E3 +61009.732}
SPL {X  -160.000, Y  +471.977, Z    +0.000, E1   -70.792, E3 +61026.251}
SPL {X  -159.977, Y  +677.138, Z    +0.000, E1   -73.665, E3 +61122.742}
SPL {X  -157.805, Y  +700.810, Z    +0.000, E1   -73.511, E3 +61139.572}
SPL {X  -152.242, Y  +723.618, Z    +0.000, E1   -72.940, E3 +61159.485}
SPL {X  -145.929, Y  +740.010, Z    +0.000, E1   -72.229, E3 +61175.957}
SPL {X  -139.114, Y  +753.439, Z    +0.000, E1   -71.436, E3 +61190.595}
SPL {X  -132.333, Y  +764.333, Z    +0.000, E1   -70.535, E3 +61203.219}
SPL {X  -125.486, Y  +773.664, Z    +0.000, E1   -69.598, E3 +61214.193}
SPL {X  -121.321, Y  +778.713, Z    +0.000, E1   -68.872, E3 +61220.203}
SPL {X   -77.337, Y  +814.468, Z    +0.000, E1   -56.377, E3 +61338.835}
ENDSPLINE

SPLINE
SPL {X  -134.727, Y  +760.706, Z    +0.000, E1   -50.460, E3 +61527.066}
SPL {X  -155.580, Y  +711.748, Z    +0.000, E1   -32.084, E3 +61543.981}
SPL {X  -159.445, Y  +687.715, Z    +0.000, E1   -14.660, E3 +61546.828}
SPL {X  -159.995, Y  +675.725, Z    +0.000, E1    -3.424, E3 +61547.339}
SPL {X  -160.000, Y  +671.714, Z    +0.000, E1    +0.835, E3 +61547.379}
SPL {X  -160.000, Y  +663.084, Z    +0.000, E1   +21.134, E3 +61547.703}
SPL {X  -160.000, Y  +650.910, Z    +0.000, E1   +46.005, E3 +61548.857}
SPL {X  -160.000, Y  +634.843, Z    +0.000, E1   +61.273, E3 +61551.534}
SPL {X  -160.000, Y  +578.679, Z    +0.000, E1   +71.665, E3 +61569.368}
SPL {X  -160.000, Y  +387.528, Z    +0.000, E1   +73.487, E3 +61662.180}
SPL {X  -159.218, Y  +369.903, Z    +0.000, E1   +73.425, E3 +61674.047}
SPL {X  -156.808, Y  +353.900, Z    +0.000, E1   +73.180, E3 +61686.651}
SPL {X  -154.539, Y  +344.254, Z    +0.000, E1   +72.827, E3 +61696.188}
ENDSPLINE

SPLINE
SPL {X  -157.258, Y  +356.206, Z    +0.000, E1   +70.434, E3 +61710.761}
ENDSPLINE

SPLINE
SPL {X  -150.342, Y  +330.952, Z    +0.000, E1   +71.154, E3 +61722.433}
SPL {X  -141.358, Y  +310.748, Z    +0.000, E1   +71.233, E3 +61735.139}
SPL {X  -134.330, Y  +298.778, Z    +0.000, E1   +70.323, E3 +61748.986}
SPL {X  -128.957, Y  +290.989, Z    +0.000, E1   +69.528, E3 +61758.351}
SPL {X  -124.846, Y  +285.632, Z    +0.000, E1   +68.906, E3 +61764.815}
SPL {X  -121.783, Y  +281.927, Z    +0.000, E1   +68.403, E3 +61769.247}
SPL {X   -79.219, Y  +246.688, Z    +0.000, E1   +55.887, E3 +61890.753}
ENDSPLINE

SPLINE
SPL {X  -125.038, Y  +285.873, Z    +0.000, E1   +53.023, E3 +62067.794}
SPL {X  -149.949, Y  +329.886, Z    +0.000, E1   +41.515, E3 +62089.359}
SPL {X  -157.246, Y  +356.141, Z    +0.000, E1   +27.282, E3 +62094.416}
SPL {X  -159.525, Y  +373.376, Z    +0.000, E1   +13.812, E3 +62096.073}
SPL {X  -160.000, Y  +387.264, Z    +0.000, E1    +0.544, E3 +62096.531}
SPL {X  -160.000, Y  +390.384, Z    +0.000, E1    -6.008, E3 +62096.568}
SPL {X  -160.000, Y  +395.752, Z    +0.000, E1   -19.038, E3 +62096.762}
SPL {X  -160.000, Y  +404.289, Z    +0.000, E1   -38.292, E3 +62097.430}
SPL {X  -160.000, Y  +418.681, Z    +0.000, E1   -56.949, E3 +62099.620}
SPL {X  -160.000, Y  +471.977, Z    +0.000, E1   -70.792, E3 +62116.139}
SPL {X  -159.977, Y  +677.138, Z    +0.000, E1   -73.665, E3 +62212.630}
SPL {X  -157.805, Y  +700.810, Z    +0.000, E1   -73.511, E3 +62229.460}
SPL {X  -152.242, Y  +723.618, Z    +0.000, E1   -72.940, E3 +62249.373}
SPL {X  -145.929, Y  +740.010, Z    +0.000, E1   -72.229, E3 +62265.845}
SPL {X  -139.114, Y  +753.439, Z    +0.000, E1   -71.436, E3 +62280.483}
SPL {X  -132.333, Y  +764.333, Z    +0.000, E1   -70.535, E3 +62293.107}
SPL {X  -125.486, Y  +773.664, Z    +0.000, E1   -69.598, E3 +62304.081}
SPL {X  -121.321, Y  +778.713, Z    +0.000, E1   -68.872, E3 +62310.091}
SPL {X   -77.337, Y  +814.468, Z    +0.000, E1   -56.377, E3 +62428.723}
ENDSPLINE

SPLINE
SPL {X  -134.727, Y  +760.706, Z    +0.000, E1   -50.460, E3 +62616.954}
SPL {X  -155.580, Y  +711.748, Z    +0.000, E1   -32.084, E3 +62633.869}
SPL {X  -159.445, Y  +687.715, Z    +0.000, E1   -14.660, E3 +62636.716}
SPL {X  -159.995, Y  +675.725, Z    +0.000, E1    -3.424, E3 +62637.227}
SPL {X  -160.000, Y  +671.714, Z    +0.000, E1    +0.835, E3 +62637.267}
SPL {X  -160.000, Y  +663.084, Z    +0.000, E1   +21.134, E3 +62637.591}
SPL {X  -160.000, Y  +650.910, Z    +0.000, E1   +46.005, E3 +62638.745}
SPL {X  -160.000, Y  +634.843, Z    +0.000, E1   +61.273, E3 +62641.422}
SPL {X  -160.000, Y  +578.679, Z    +0.000, E1   +71.665, E3 +62659.256}
SPL {X  -160.000, Y  +387.528, Z    +0.000, E1   +73.487, E3 +62752.068}
SPL {X  -159.218, Y  +369.903, Z    +0.000, E1   +73.425, E3 +62763.935}
SPL {X  -156.808, Y  +353.900, Z    +0.000, E1   +73.180, E3 +62776.539}
SPL {X  -154.539, Y  +344.254, Z    +0.000, E1   +72.827, E3 +62786.076}
ENDSPLINE

SPLINE
SPL {X  -157.258, Y  +356.206, Z    +0.000, E1   +70.434, E3 +62800.649}
ENDSPLINE

SPLINE
SPL {X  -150.342, Y  +330.952, Z    +0.000, E1   +71.154, E3 +62812.321}
SPL {X  -141.358, Y  +310.748, Z    +0.000, E1   +71.233, E3 +62825.027}
SPL {X  -134.330, Y  +298.778, Z    +0.000, E1   +70.323, E3 +62838.874}
SPL {X  -128.957, Y  +290.989, Z    +0.000, E1   +69.528, E3 +62848.239}
SPL {X  -124.846, Y  +285.632, Z    +0.000, E1   +68.906, E3 +62854.703}
SPL {X  -121.783, Y  +281.927, Z    +0.000, E1   +68.403, E3 +62859.135}
SPL {X   -79.219, Y  +246.688, Z    +0.000, E1   +55.887, E3 +62980.641}
ENDSPLINE

SPLINE
SPL {X  -125.038, Y  +285.873, Z    +0.000, E1   +53.023, E3 +63157.682}
SPL {X  -149.949, Y  +329.886, Z    +0.000, E1   +41.515, E3 +63179.247}
SPL {X  -157.246, Y  +356.141, Z    +0.000, E1   +27.282, E3 +63184.304}
SPL {X  -159.525, Y  +373.376, Z    +0.000, E1   +13.812, E3 +63185.961}
SPL {X  -160.000, Y  +387.264, Z    +0.000, E1    +0.544, E3 +63186.419}
SPL {X  -160.000, Y  +390.384, Z    +0.000, E1    -6.008, E3 +63186.456}
SPL {X  -160.000, Y  +395.752, Z    +0.000, E1   -19.038, E3 +63186.650}
SPL {X  -160.000, Y  +404.289, Z    +0.000, E1   -38.292, E3 +63187.318}
SPL {X  -160.000, Y  +418.681, Z    +0.000, E1   -56.949, E3 +63189.508}
SPL {X  -160.000, Y  +471.977, Z    +0.000, E1   -70.792, E3 +63206.027}
SPL {X  -159.977, Y  +677.138, Z    +0.000, E1   -73.665, E3 +63302.518}
SPL {X  -157.805, Y  +700.810, Z    +0.000, E1   -73.511, E3 +63319.348}
SPL {X  -152.242, Y  +723.618, Z    +0.000, E1   -72.940, E3 +63339.261}
SPL {X  -145.929, Y  +740.010, Z    +0.000, E1   -72.229, E3 +63355.733}
SPL {X  -139.114, Y  +753.439, Z    +0.000, E1   -71.436, E3 +63370.371}
SPL {X  -132.333, Y  +764.333, Z    +0.000, E1   -70.535, E3 +63382.995}
SPL {X  -125.486, Y  +773.664, Z    +0.000, E1   -69.598, E3 +63393.969}
SPL {X  -121.321, Y  +778.713, Z    +0.000, E1   -68.872, E3 +63399.979}
SPL {X   -77.337, Y  +814.468, Z    +0.000, E1   -56.377, E3 +63518.611}
ENDSPLINE

SPLINE
SPL {X  -134.727, Y  +760.706, Z    +0.000, E1   -50.460, E3 +63706.842}
SPL {X  -155.580, Y  +711.748, Z    +0.000, E1   -32.084, E3 +63723.757}
SPL {X  -159.445, Y  +687.715, Z    +0.000, E1   -14.660, E3 +63726.604}
SPL {X  -159.995, Y  +675.725, Z    +0.000, E1    -3.424, E3 +63727.115}
SPL {X  -160.000, Y  +671.714, Z    +0.000, E1    +0.835, E3 +63727.155}
SPL {X  -160.000, Y  +663.084, Z    +0.000, E1   +21.134, E3 +63727.479}
SPL {X  -160.000, Y  +650.910, Z    +0.000, E1   +46.005, E3 +63728.633}
SPL {X  -160.000, Y  +634.843, Z    +0.000, E1   +61.273, E3 +63731.310}
SPL {X  -160.000, Y  +578.679, Z    +0.000, E1   +71.665, E3 +63749.144}
SPL {X  -160.000, Y  +387.528, Z    +0.000, E1   +73.487, E3 +63841.956}
SPL {X  -159.218, Y  +369.903, Z    +0.000, E1   +73.425, E3 +63853.823}
SPL {X  -156.808, Y  +353.900, Z    +0.000, E1   +73.180, E3 +63866.427}
SPL {X  -154.539, Y  +344.254, Z    +0.000, E1   +72.827, E3 +63875.964}
ENDSPLINE

SPLINE
SPL {X  -157.258, Y  +356.206, Z    +0.000, E1   +70.434, E3 +63890.537}
ENDSPLINE

SPLINE
SPL {X  -150.342, Y  +330.952, Z    +0.000, E1   +71.154, E3 +63902.209}
SPL {X  -141.358, Y  +310.748, Z    +0.000, E1   +71.233, E3 +63914.915}
SPL {X  -134.330, Y  +298.778, Z    +0.000, E1   +70.323, E3 +63928.762}
SPL {X  -128.957, Y  +290.989, Z    +0.000, E1   +69.528, E3 +63938.127}
SPL {X  -124.846, Y  +285.632, Z    +0.000, E1   +68.906, E3 +63944.591}
SPL {X  -121.783, Y  +281.927, Z    +0.000, E1   +68.403, E3 +63949.023}
SPL {X   -79.219, Y  +246.688, Z    +0.000, E1   +55.887, E3 +64070.529}
ENDSPLINE

SPLINE
SPL {X  -125.038, Y  +285.873, Z    +0.000, E1   +53.023, E3 +64247.570}
SPL {X  -149.949, Y  +329.886, Z    +0.000, E1   +41.515, E3 +64269.135}
SPL {X  -157.246, Y  +356.141, Z    +0.000, E1   +27.282, E3 +64274.192}
SPL {X  -159.525, Y  +373.376, Z    +0.000, E1   +13.812, E3 +64275.849}
SPL {X  -160.000, Y  +387.264, Z    +0.000, E1    +0.544, E3 +64276.307}
SPL {X  -160.000, Y  +390.384, Z    +0.000, E1    -6.008, E3 +64276.344}
SPL {X  -160.000, Y  +395.752, Z    +0.000, E1   -19.038, E3 +64276.538}
SPL {X  -160.000, Y  +404.289, Z    +0.000, E1   -38.292, E3 +64277.206}
SPL {X  -160.000, Y  +418.681, Z    +0.000, E1   -56.949, E3 +64279.396}
SPL {X  -160.000, Y  +458.961, Z    +0.000, E1   -69.778, E3 +64290.992}
SPL {X  -160.000, Y  +485.343, Z    +0.000, E1   -71.539, E3 +64300.978}
SPL {X  -159.977, Y  +677.138, Z    +0.000, E1   -73.665, E3 +64392.406}
SPL {X  -157.805, Y  +700.810, Z    +0.000, E1   -73.511, E3 +64409.237}
SPL {X  -152.242, Y  +723.618, Z    +0.000, E1   -72.940, E3 +64429.149}
SPL {X  -145.929, Y  +740.010, Z    +0.000, E1   -72.229, E3 +64445.621}
SPL {X  -139.114, Y  +753.439, Z    +0.000, E1   -71.436, E3 +64460.259}
SPL {X  -132.333, Y  +764.333, Z    +0.000, E1   -70.535, E3 +64472.883}
SPL {X  -125.486, Y  +773.664, Z    +0.000, E1   -69.598, E3 +64483.857}
SPL {X  -121.321, Y  +778.713, Z    +0.000, E1   -68.872, E3 +64489.867}
SPL {X   -77.337, Y  +814.468, Z    +0.000, E1   -56.377, E3 +64608.499}
ENDSPLINE

SPLINE
SPL {X  -134.727, Y  +760.706, Z    +0.000, E1   -50.460, E3 +64796.731}
SPL {X  -155.580, Y  +711.748, Z    +0.000, E1   -32.084, E3 +64813.645}
SPL {X  -159.445, Y  +687.715, Z    +0.000, E1   -14.660, E3 +64816.492}
SPL {X  -159.995, Y  +675.725, Z    +0.000, E1    -3.424, E3 +64817.003}
SPL {X  -160.000, Y  +671.714, Z    +0.000, E1    +0.835, E3 +64817.043}
SPL {X  -160.000, Y  +663.084, Z    +0.000, E1   +21.134, E3 +64817.368}
SPL {X  -160.000, Y  +650.910, Z    +0.000, E1   +46.005, E3 +64818.521}
SPL {X  -160.000, Y  +634.843, Z    +0.000, E1   +61.273, E3 +64821.198}
SPL {X  -160.000, Y  +578.679, Z    +0.000, E1   +71.665, E3 +64839.032}
SPL {X  -160.000, Y  +387.528, Z    +0.000, E1   +73.487, E3 +64931.844}
SPL {X  -159.218, Y  +369.903, Z    +0.000, E1   +73.425, E3 +64943.711}
SPL {X  -156.808, Y  +353.900, Z    +0.000, E1   +73.180, E3 +64956.315}
SPL {X  -154.539, Y  +344.254, Z    +0.000, E1   +72.827, E3 +64965.853}
ENDSPLINE

SPLINE
SPL {X  -157.258, Y  +356.206, Z    +0.000, E1   +70.434, E3 +64980.425}
ENDSPLINE

SPLINE
SPL {X  -150.342, Y  +330.952, Z    +0.000, E1   +71.154, E3 +64992.097}
SPL {X  -141.358, Y  +310.748, Z    +0.000, E1   +71.233, E3 +65004.803}
SPL {X  -134.330, Y  +298.778, Z    +0.000, E1   +70.323, E3 +65018.650}
SPL {X  -128.957, Y  +290.989, Z    +0.000, E1   +69.528, E3 +65028.016}
SPL {X  -124.846, Y  +285.632, Z    +0.000, E1   +68.906, E3 +65034.479}
SPL {X  -121.783, Y  +281.927, Z    +0.000, E1   +68.403, E3 +65038.911}
SPL {X   -79.219, Y  +246.688, Z    +0.000, E1   +55.887, E3 +65160.417}
ENDSPLINE

SPLINE
SPL {X  -125.038, Y  +285.873, Z    +0.000, E1   +53.023, E3 +65337.458}
SPL {X  -149.949, Y  +329.886, Z    +0.000, E1   +41.515, E3 +65359.024}
SPL {X  -157.246, Y  +356.141, Z    +0.000, E1   +27.282, E3 +65364.080}
SPL {X  -159.525, Y  +373.376, Z    +0.000, E1   +13.812, E3 +65365.737}
SPL {X  -160.000, Y  +387.264, Z    +0.000, E1    +0.544, E3 +65366.195}
SPL {X  -160.000, Y  +390.384, Z    +0.000, E1    -6.008, E3 +65366.232}
SPL {X  -160.000, Y  +395.752, Z    +0.000, E1   -19.038, E3 +65366.426}
SPL {X  -160.000, Y  +404.289, Z    +0.000, E1   -38.292, E3 +65367.094}
SPL {X  -160.000, Y  +418.681, Z    +0.000, E1   -56.949, E3 +65369.284}
SPL {X  -160.000, Y  +458.961, Z    +0.000, E1   -69.778, E3 +65380.880}
SPL {X  -160.000, Y  +485.343, Z    +0.000, E1   -71.539, E3 +65390.866}
SPL {X  -159.977, Y  +677.138, Z    +0.000, E1   -73.665, E3 +65482.294}
SPL {X  -157.805, Y  +700.810, Z    +0.000, E1   -73.511, E3 +65499.125}
SPL {X  -152.242, Y  +723.618, Z    +0.000, E1   -72.940, E3 +65519.037}
SPL {X  -145.929, Y  +740.010, Z    +0.000, E1   -72.229, E3 +65535.509}
SPL {X  -139.114, Y  +753.439, Z    +0.000, E1   -71.436, E3 +65550.147}
SPL {X  -132.333, Y  +764.333, Z    +0.000, E1   -70.535, E3 +65562.771}
SPL {X  -125.486, Y  +773.664, Z    +0.000, E1   -69.598, E3 +65573.745}
SPL {X  -121.321, Y  +778.713, Z    +0.000, E1   -68.872, E3 +65579.755}
SPL {X   -77.337, Y  +814.468, Z    +0.000, E1   -56.377, E3 +65698.387}
ENDSPLINE

SPLINE
SPL {X  -134.727, Y  +760.706, Z    +0.000, E1   -50.460, E3 +65886.619}
SPL {X  -155.580, Y  +711.748, Z    +0.000, E1   -32.084, E3 +65903.533}
SPL {X  -159.445, Y  +687.715, Z    +0.000, E1   -14.660, E3 +65906.380}
SPL {X  -159.995, Y  +675.725, Z    +0.000, E1    -3.424, E3 +65906.891}
SPL {X  -160.000, Y  +671.714, Z    +0.000, E1    +0.835, E3 +65906.931}
SPL {X  -160.000, Y  +663.084, Z    +0.000, E1   +21.134, E3 +65907.256}
SPL {X  -160.000, Y  +650.910, Z    +0.000, E1   +46.005, E3 +65908.409}
SPL {X  -160.000, Y  +634.843, Z    +0.000, E1   +61.273, E3 +65911.086}
SPL {X  -160.000, Y  +578.679, Z    +0.000, E1   +71.665, E3 +65928.920}
SPL {X  -160.000, Y  +387.528, Z    +0.000, E1   +73.487, E3 +66021.732}
SPL {X  -159.218, Y  +369.903, Z    +0.000, E1   +73.425, E3 +66033.600}
SPL {X  -156.808, Y  +353.900, Z    +0.000, E1   +73.180, E3 +66046.203}
SPL {X  -154.539, Y  +344.254, Z    +0.000, E1   +72.827, E3 +66055.741}
ENDSPLINE

SPLINE
SPL {X  -157.258, Y  +356.206, Z    +0.000, E1   +70.434, E3 +66070.313}
ENDSPLINE

SPLINE
SPL {X  -150.342, Y  +330.952, Z    +0.000, E1   +71.154, E3 +66081.985}
SPL {X  -141.358, Y  +310.748, Z    +0.000, E1   +71.233, E3 +66094.691}
SPL {X  -134.330, Y  +298.778, Z    +0.000, E1   +70.323, E3 +66108.538}
SPL {X  -128.957, Y  +290.989, Z    +0.000, E1   +69.528, E3 +66117.904}
SPL {X  -124.846, Y  +285.632, Z    +0.000, E1   +68.906, E3 +66124.367}
SPL {X  -121.783, Y  +281.927, Z    +0.000, E1   +68.403, E3 +66128.799}
SPL {X   -79.219, Y  +246.688, Z    +0.000, E1   +55.887, E3 +66250.305}
ENDSPLINE

SPLINE
SPL {X  -125.038, Y  +285.873, Z    +0.000, E1   +53.023, E3 +66427.346}
SPL {X  -149.949, Y  +329.886, Z    +0.000, E1   +41.515, E3 +66448.912}
SPL {X  -157.246, Y  +356.141, Z    +0.000, E1   +27.282, E3 +66453.968}
SPL {X  -159.525, Y  +373.376, Z    +0.000, E1   +13.812, E3 +66455.625}
SPL {X  -160.000, Y  +387.264, Z    +0.000, E1    +0.544, E3 +66456.083}
SPL {X  -160.000, Y  +390.384, Z    +0.000, E1    -6.008, E3 +66456.120}
SPL {X  -160.000, Y  +395.752, Z    +0.000, E1   -19.038, E3 +66456.314}
SPL {X  -160.000, Y  +404.289, Z    +0.000, E1   -38.292, E3 +66456.982}
SPL {X  -160.000, Y  +418.681, Z    +0.000, E1   -56.949, E3 +66459.172}
SPL {X  -160.000, Y  +471.977, Z    +0.000, E1   -70.792, E3 +66475.691}
SPL {X  -159.977, Y  +677.138, Z    +0.000, E1   -73.665, E3 +66572.182}
SPL {X  -157.805, Y  +700.810, Z    +0.000, E1   -73.511, E3 +66589.013}
SPL {X  -152.242, Y  +723.618, Z    +0.000, E1   -72.940, E3 +66608.925}
SPL {X  -145.929, Y  +740.010, Z    +0.000, E1   -72.229, E3 +66625.397}
SPL {X  -139.114, Y  +753.439, Z    +0.000, E1   -71.436, E3 +66640.035}
SPL {X  -132.333, Y  +764.333, Z    +0.000, E1   -70.535, E3 +66652.659}
SPL {X  -125.486, Y  +773.664, Z    +0.000, E1   -69.598, E3 +66663.633}
SPL {X  -121.321, Y  +778.713, Z    +0.000, E1   -68.872, E3 +66669.643}
SPL {X   -77.337, Y  +814.468, Z    +0.000, E1   -56.377, E3 +66788.275}
ENDSPLINE

SPLINE
SPL {X  -134.727, Y  +760.706, Z    +0.000, E1   -50.460, E3 +66976.507}
SPL {X  -155.580, Y  +711.748, Z    +0.000, E1   -32.084, E3 +66993.421}
SPL {X  -159.445, Y  +687.715, Z    +0.000, E1   -14.660, E3 +66996.268}
SPL {X  -159.995, Y  +675.725, Z    +0.000, E1    -3.424, E3 +66996.779}
SPL {X  -160.000, Y  +671.714, Z    +0.000, E1    +0.835, E3 +66996.819}
SPL {X  -160.000, Y  +663.084, Z    +0.000, E1   +21.134, E3 +66997.144}
SPL {X  -160.000, Y  +650.910, Z    +0.000, E1   +46.005, E3 +66998.297}
SPL {X  -160.000, Y  +634.843, Z    +0.000, E1   +61.273, E3 +67000.974}
SPL {X  -160.000, Y  +578.679, Z    +0.000, E1   +71.665, E3 +67018.808}
SPL {X  -160.000, Y  +387.528, Z    +0.000, E1   +73.487, E3 +67111.620}
SPL {X  -159.218, Y  +369.903, Z    +0.000, E1   +73.425, E3 +67123.488}
SPL {X  -156.808, Y  +353.900, Z    +0.000, E1   +73.180, E3 +67136.091}
SPL {X  -154.539, Y  +344.254, Z    +0.000, E1   +72.827, E3 +67145.629}
ENDSPLINE

SPLINE
SPL {X  -157.258, Y  +356.206, Z    +0.000, E1   +70.434, E3 +67160.201}
ENDSPLINE

SPLINE
SPL {X  -150.342, Y  +330.952, Z    +0.000, E1   +71.154, E3 +67171.873}
SPL {X  -141.358, Y  +310.748, Z    +0.000, E1   +71.233, E3 +67184.579}
SPL {X  -134.330, Y  +298.778, Z    +0.000, E1   +70.323, E3 +67198.426}
SPL {X  -128.957, Y  +290.989, Z    +0.000, E1   +69.528, E3 +67207.792}
SPL {X  -124.846, Y  +285.632, Z    +0.000, E1   +68.906, E3 +67214.255}
SPL {X  -121.783, Y  +281.927, Z    +0.000, E1   +68.403, E3 +67218.687}
SPL {X   -79.219, Y  +246.688, Z    +0.000, E1   +55.887, E3 +67340.193}
ENDSPLINE

SPLINE
SPL {X  -125.038, Y  +285.873, Z    +0.000, E1   +53.023, E3 +67517.235}
SPL {X  -149.949, Y  +329.886, Z    +0.000, E1   +41.515, E3 +67538.800}
SPL {X  -157.246, Y  +356.141, Z    +0.000, E1   +27.282, E3 +67543.856}
SPL {X  -159.525, Y  +373.376, Z    +0.000, E1   +13.812, E3 +67545.513}
SPL {X  -160.000, Y  +387.264, Z    +0.000, E1    +0.544, E3 +67545.971}
SPL {X  -160.000, Y  +390.384, Z    +0.000, E1    -6.008, E3 +67546.008}
SPL {X  -160.000, Y  +395.752, Z    +0.000, E1   -19.038, E3 +67546.202}
SPL {X  -160.000, Y  +404.289, Z    +0.000, E1   -38.292, E3 +67546.870}
SPL {X  -160.000, Y  +418.681, Z    +0.000, E1   -56.949, E3 +67549.060}
SPL {X  -160.000, Y  +471.977, Z    +0.000, E1   -70.792, E3 +67565.579}
SPL {X  -159.977, Y  +677.138, Z    +0.000, E1   -73.665, E3 +67662.070}
SPL {X  -157.805, Y  +700.810, Z    +0.000, E1   -73.511, E3 +67678.901}
SPL {X  -152.242, Y  +723.618, Z    +0.000, E1   -72.940, E3 +67698.814}
SPL {X  -145.929, Y  +740.010, Z    +0.000, E1   -72.229, E3 +67715.285}
SPL {X  -139.114, Y  +753.439, Z    +0.000, E1   -71.436, E3 +67729.924}
SPL {X  -132.333, Y  +764.333, Z    +0.000, E1   -70.535, E3 +67742.547}
SPL {X  -125.486, Y  +773.664, Z    +0.000, E1   -69.598, E3 +67753.522}
SPL {X  -121.321, Y  +778.713, Z    +0.000, E1   -68.872, E3 +67759.532}
SPL {X   -77.337, Y  +814.468, Z    +0.000, E1   -56.377, E3 +67878.163}
ENDSPLINE

SPLINE
SPL {X  -134.727, Y  +760.706, Z    +0.000, E1   -50.460, E3 +68066.395}
SPL {X  -155.580, Y  +711.748, Z    +0.000, E1   -32.084, E3 +68083.309}
SPL {X  -159.445, Y  +687.715, Z    +0.000, E1   -14.660, E3 +68086.156}
SPL {X  -159.995, Y  +675.725, Z    +0.000, E1    -3.424, E3 +68086.667}
SPL {X  -160.000, Y  +671.714, Z    +0.000, E1    +0.835, E3 +68086.707}
SPL {X  -160.000, Y  +663.084, Z    +0.000, E1   +21.134, E3 +68087.032}
SPL {X  -160.000, Y  +650.910, Z    +0.000, E1   +46.005, E3 +68088.185}
SPL {X  -160.000, Y  +634.843, Z    +0.000, E1   +61.273, E3 +68090.862}
SPL {X  -160.000, Y  +578.679, Z    +0.000, E1   +71.665, E3 +68108.696}
SPL {X  -160.000, Y  +387.528, Z    +0.000, E1   +73.487, E3 +68201.508}
SPL {X  -159.218, Y  +369.903, Z    +0.000, E1   +73.425, E3 +68213.376}
SPL {X  -156.808, Y  +353.900, Z    +0.000, E1   +73.180, E3 +68225.979}
SPL {X  -154.539, Y  +344.254, Z    +0.000, E1   +72.827, E3 +68235.517}
ENDSPLINE

SPLINE
SPL {X  -157.258, Y  +356.206, Z    +0.000, E1   +70.434, E3 +68250.089}
ENDSPLINE

SPLINE
SPL {X  -150.342, Y  +330.952, Z    +0.000, E1   +71.154, E3 +68261.761}
SPL {X  -141.358, Y  +310.748, Z    +0.000, E1   +71.233, E3 +68274.467}
SPL {X  -134.330, Y  +298.778, Z    +0.000, E1   +70.323, E3 +68288.314}
SPL {X  -128.957, Y  +290.989, Z    +0.000, E1   +69.528, E3 +68297.680}
SPL {X  -124.846, Y  +285.632, Z    +0.000, E1   +68.906, E3 +68304.143}
SPL {X  -121.783, Y  +281.927, Z    +0.000, E1   +68.403, E3 +68308.575}
SPL {X   -79.219, Y  +246.688, Z    +0.000, E1   +55.887, E3 +68430.081}
ENDSPLINE

SPLINE
SPL {X  -125.038, Y  +285.873, Z    +0.000, E1   +53.023, E3 +68607.123}
SPL {X  -149.949, Y  +329.886, Z    +0.000, E1   +41.515, E3 +68628.688}
SPL {X  -157.246, Y  +356.141, Z    +0.000, E1   +27.282, E3 +68633.744}
SPL {X  -159.525, Y  +373.376, Z    +0.000, E1   +13.812, E3 +68635.401}
SPL {X  -160.000, Y  +387.264, Z    +0.000, E1    +0.544, E3 +68635.859}
SPL {X  -160.000, Y  +390.384, Z    +0.000, E1    -6.008, E3 +68635.896}
SPL {X  -160.000, Y  +395.752, Z    +0.000, E1   -19.038, E3 +68636.090}
SPL {X  -160.000, Y  +404.289, Z    +0.000, E1   -38.292, E3 +68636.758}
SPL {X  -160.000, Y  +418.681, Z    +0.000, E1   -56.949, E3 +68638.948}
SPL {X  -160.000, Y  +471.977, Z    +0.000, E1   -70.792, E3 +68655.467}
SPL {X  -159.977, Y  +677.138, Z    +0.000, E1   -73.665, E3 +68751.958}
SPL {X  -157.805, Y  +700.810, Z    +0.000, E1   -73.511, E3 +68768.789}
SPL {X  -152.242, Y  +723.618, Z    +0.000, E1   -72.940, E3 +68788.702}
SPL {X  -145.929, Y  +740.010, Z    +0.000, E1   -72.229, E3 +68805.173}
SPL {X  -139.114, Y  +753.439, Z    +0.000, E1   -71.436, E3 +68819.812}
SPL {X  -132.333, Y  +764.333, Z    +0.000, E1   -70.535, E3 +68832.435}
SPL {X  -125.486, Y  +773.664, Z    +0.000, E1   -69.598, E3 +68843.410}
SPL {X  -121.321, Y  +778.713, Z    +0.000, E1   -68.872, E3 +68849.420}
SPL {X   -77.337, Y  +814.468, Z    +0.000, E1   -56.377, E3 +68968.051}
ENDSPLINE

SPLINE
SPL {X  -134.727, Y  +760.706, Z    +0.000, E1   -50.460, E3 +69156.283}
SPL {X  -155.580, Y  +711.748, Z    +0.000, E1   -32.084, E3 +69173.197}
SPL {X  -159.445, Y  +687.715, Z    +0.000, E1   -14.660, E3 +69176.044}
SPL {X  -159.995, Y  +675.725, Z    +0.000, E1    -3.424, E3 +69176.555}
SPL {X  -160.000, Y  +671.714, Z    +0.000, E1    +0.835, E3 +69176.595}
SPL {X  -160.000, Y  +663.084, Z    +0.000, E1   +21.134, E3 +69176.920}
SPL {X  -160.000, Y  +650.910, Z    +0.000, E1   +46.005, E3 +69178.073}
SPL {X  -160.000, Y  +634.843, Z    +0.000, E1   +61.273, E3 +69180.750}
SPL {X  -160.000, Y  +578.679, Z    +0.000, E1   +71.665, E3 +69198.584}
SPL {X  -160.000, Y  +387.528, Z    +0.000, E1   +73.487, E3 +69291.396}
SPL {X  -159.218, Y  +369.903, Z    +0.000, E1   +73.425, E3 +69303.264}
SPL {X  -156.808, Y  +353.900, Z    +0.000, E1   +73.180, E3 +69315.867}
SPL {X  -154.539, Y  +344.254, Z    +0.000, E1   +72.827, E3 +69325.405}
ENDSPLINE

SPLINE
SPL {X  -157.258, Y  +356.206, Z    +0.000, E1   +70.434, E3 +69339.977}
ENDSPLINE

SPLINE
SPL {X  -150.342, Y  +330.952, Z    +0.000, E1   +71.154, E3 +69351.649}
SPL {X  -141.358, Y  +310.748, Z    +0.000, E1   +71.233, E3 +69364.355}
SPL {X  -134.330, Y  +298.778, Z    +0.000, E1   +70.323, E3 +69378.202}
SPL {X  -128.957, Y  +290.989, Z    +0.000, E1   +69.528, E3 +69387.568}
SPL {X  -124.846, Y  +285.632, Z    +0.000, E1   +68.906, E3 +69394.031}
SPL {X  -121.783, Y  +281.927, Z    +0.000, E1   +68.403, E3 +69398.463}
SPL {X   -79.219, Y  +246.688, Z    +0.000, E1   +55.887, E3 +69519.969}
ENDSPLINE

SPLINE
SPL {X  -125.038, Y  +285.873, Z    +0.000, E1   +53.023, E3 +69697.011}
SPL {X  -149.949, Y  +329.886, Z    +0.000, E1   +41.515, E3 +69718.576}
SPL {X  -157.246, Y  +356.141, Z    +0.000, E1   +27.282, E3 +69723.632}
SPL {X  -159.525, Y  +373.376, Z    +0.000, E1   +13.812, E3 +69725.289}
SPL {X  -160.000, Y  +387.264, Z    +0.000, E1    +0.544, E3 +69725.747}
SPL {X  -160.000, Y  +390.384, Z    +0.000, E1    -6.008, E3 +69725.784}
SPL {X  -160.000, Y  +395.752, Z    +0.000, E1   -19.038, E3 +69725.978}
SPL {X  -160.000, Y  +404.289, Z    +0.000, E1   -38.292, E3 +69726.646}
SPL {X  -160.000, Y  +418.681, Z    +0.000, E1   -56.949, E3 +69728.836}
SPL {X  -160.000, Y  +471.977, Z    +0.000, E1   -70.792, E3 +69745.355}
SPL {X  -159.977, Y  +677.138, Z    +0.000, E1   -73.665, E3 +69841.847}
SPL {X  -157.805, Y  +700.810, Z    +0.000, E1   -73.511, E3 +69858.677}
SPL {X  -152.242, Y  +723.618, Z    +0.000, E1   -72.940, E3 +69878.590}
SPL {X  -145.929, Y  +740.010, Z    +0.000, E1   -72.229, E3 +69895.061}
SPL {X  -139.114, Y  +753.439, Z    +0.000, E1   -71.436, E3 +69909.700}
SPL {X  -132.333, Y  +764.333, Z    +0.000, E1   -70.535, E3 +69922.323}
SPL {X  -125.486, Y  +773.664, Z    +0.000, E1   -69.598, E3 +69933.298}
SPL {X  -121.321, Y  +778.713, Z    +0.000, E1   -68.872, E3 +69939.308}
SPL {X   -77.337, Y  +814.468, Z    +0.000, E1   -56.377, E3 +70057.939}
ENDSPLINE

SPLINE
SPL {X  -134.727, Y  +760.706, Z    +0.000, E1   -50.460, E3 +70246.171}
SPL {X  -155.580, Y  +711.748, Z    +0.000, E1   -32.084, E3 +70263.085}
SPL {X  -159.445, Y  +687.715, Z    +0.000, E1   -14.660, E3 +70265.932}
SPL {X  -159.995, Y  +675.725, Z    +0.000, E1    -3.424, E3 +70266.443}
SPL {X  -160.000, Y  +671.714, Z    +0.000, E1    +0.835, E3 +70266.483}
SPL {X  -160.000, Y  +663.084, Z    +0.000, E1   +21.134, E3 +70266.808}
SPL {X  -160.000, Y  +650.910, Z    +0.000, E1   +46.005, E3 +70267.961}
SPL {X  -160.000, Y  +634.843, Z    +0.000, E1   +61.273, E3 +70270.638}
SPL {X  -160.000, Y  +578.679, Z    +0.000, E1   +71.665, E3 +70288.472}
SPL {X  -160.000, Y  +387.528, Z    +0.000, E1   +73.487, E3 +70381.284}
SPL {X  -159.218, Y  +369.903, Z    +0.000, E1   +73.425, E3 +70393.152}
SPL {X  -156.808, Y  +353.900, Z    +0.000, E1   +73.180, E3 +70405.755}
SPL {X  -154.539, Y  +344.254, Z    +0.000, E1   +72.827, E3 +70415.293}
ENDSPLINE

SPLINE
SPL {X  -157.258, Y  +356.206, Z    +0.000, E1   +70.434, E3 +70429.865}
ENDSPLINE

SPLINE
SPL {X  -150.342, Y  +330.952, Z    +0.000, E1   +71.154, E3 +70441.538}
SPL {X  -141.358, Y  +310.748, Z    +0.000, E1   +71.233, E3 +70454.243}
SPL {X  -134.330, Y  +298.778, Z    +0.000, E1   +70.323, E3 +70468.090}
SPL {X  -128.957, Y  +290.989, Z    +0.000, E1   +69.528, E3 +70477.456}
SPL {X  -124.846, Y  +285.632, Z    +0.000, E1   +68.906, E3 +70483.919}
SPL {X  -121.783, Y  +281.927, Z    +0.000, E1   +68.403, E3 +70488.351}
SPL {X   -79.219, Y  +246.688, Z    +0.000, E1   +55.887, E3 +70609.858}
ENDSPLINE

SPLINE
SPL {X  -125.038, Y  +285.873, Z    +0.000, E1   +53.023, E3 +70786.899}
SPL {X  -149.949, Y  +329.886, Z    +0.000, E1   +41.515, E3 +70808.464}
SPL {X  -157.246, Y  +356.141, Z    +0.000, E1   +27.282, E3 +70813.520}
SPL {X  -159.525, Y  +373.376, Z    +0.000, E1   +13.812, E3 +70815.177}
SPL {X  -160.000, Y  +387.264, Z    +0.000, E1    +0.544, E3 +70815.635}
SPL {X  -160.000, Y  +390.384, Z    +0.000, E1    -6.008, E3 +70815.672}
SPL {X  -160.000, Y  +395.752, Z    +0.000, E1   -19.038, E3 +70815.866}
SPL {X  -160.000, Y  +404.289, Z    +0.000, E1   -38.292, E3 +70816.534}
SPL {X  -160.000, Y  +418.681, Z    +0.000, E1   -56.949, E3 +70818.724}
SPL {X  -160.000, Y  +471.977, Z    +0.000, E1   -70.792, E3 +70835.243}
SPL {X  -159.977, Y  +677.138, Z    +0.000, E1   -73.665, E3 +70931.735}
SPL {X  -157.805, Y  +700.810, Z    +0.000, E1   -73.511, E3 +70948.565}
SPL {X  -152.242, Y  +723.618, Z    +0.000, E1   -72.940, E3 +70968.478}
SPL {X  -145.929, Y  +740.010, Z    +0.000, E1   -72.229, E3 +70984.949}
SPL {X  -139.114, Y  +753.439, Z    +0.000, E1   -71.436, E3 +70999.588}
SPL {X  -132.333, Y  +764.333, Z    +0.000, E1   -70.535, E3 +71012.211}
SPL {X  -125.486, Y  +773.664, Z    +0.000, E1   -69.598, E3 +71023.186}
SPL {X  -121.321, Y  +778.713, Z    +0.000, E1   -68.872, E3 +71029.196}
SPL {X   -77.337, Y  +814.468, Z    +0.000, E1   -56.377, E3 +71147.827}
ENDSPLINE

SPLINE
SPL {X  -134.727, Y  +760.706, Z    +0.000, E1   -50.460, E3 +71336.059}
SPL {X  -155.580, Y  +711.748, Z    +0.000, E1   -32.084, E3 +71352.973}
SPL {X  -159.445, Y  +687.715, Z    +0.000, E1   -14.660, E3 +71355.820}
SPL {X  -159.995, Y  +675.725, Z    +0.000, E1    -3.424, E3 +71356.331}
SPL {X  -160.000, Y  +671.714, Z    +0.000, E1    +0.835, E3 +71356.371}
SPL {X  -160.000, Y  +663.084, Z    +0.000, E1   +21.134, E3 +71356.696}
SPL {X  -160.000, Y  +650.910, Z    +0.000, E1   +46.005, E3 +71357.849}
SPL {X  -160.000, Y  +634.843, Z    +0.000, E1   +61.273, E3 +71360.526}
SPL {X  -160.000, Y  +578.679, Z    +0.000, E1   +71.665, E3 +71378.360}
SPL {X  -160.000, Y  +387.528, Z    +0.000, E1   +73.487, E3 +71471.172}
SPL {X  -159.218, Y  +369.903, Z    +0.000, E1   +73.425, E3 +71483.040}
SPL {X  -156.808, Y  +353.900, Z    +0.000, E1   +73.180, E3 +71495.643}
SPL {X  -154.539, Y  +344.254, Z    +0.000, E1   +72.827, E3 +71505.181}
ENDSPLINE

SPLINE
SPL {X  -157.258, Y  +356.206, Z    +0.000, E1   +70.434, E3 +71519.753}
ENDSPLINE

SPLINE
SPL {X  -150.342, Y  +330.952, Z    +0.000, E1   +71.154, E3 +71531.426}
SPL {X  -141.358, Y  +310.748, Z    +0.000, E1   +71.233, E3 +71544.131}
SPL {X  -134.330, Y  +298.778, Z    +0.000, E1   +70.323, E3 +71557.979}
SPL {X  -128.957, Y  +290.989, Z    +0.000, E1   +69.528, E3 +71567.344}
SPL {X  -124.846, Y  +285.632, Z    +0.000, E1   +68.906, E3 +71573.807}
SPL {X  -121.783, Y  +281.927, Z    +0.000, E1   +68.403, E3 +71578.239}
SPL {X   -79.219, Y  +246.688, Z    +0.000, E1   +55.887, E3 +71699.746}
ENDSPLINE

